ORGANIZATION_BLOCK OB 1
TITLE = "Main Program Sweep (Cycle)"
AUTHOR : Kng
NAME : Main
VERSION : 0.1
VAR_TEMP
  OB1_EV_CLASS : BYTE ;	//Bits 0-3 = 1 (Coming event), Bits 4-7 = 1 (Event class 1)
  OB1_SCAN_1 : BYTE ;	//1 (Cold restart scan 1 of OB 1), 3 (Scan 2-n of OB 1)
  OB1_PRIORITY : BYTE ;	//Priority of OB Execution
  OB1_OB_NUMBR : BYTE ;	//1 (Organization block 1, OB1)
  OB1_RESERVED_1 : BYTE ;	//Reserved for system
  OB1_RESERVED_2 : BYTE ;	//Reserved for system
  OB1_PREV_CYCLE : INT ;	//Cycle time of previous OB1 scan (milliseconds)
  OB1_MIN_CYCLE : INT ;	//Minimum cycle time of OB1 (milliseconds)
  OB1_MAX_CYCLE : INT ;	//Maximum cycle time of OB1 (milliseconds)
  OB1_DATE_TIME : DATE_AND_TIME ;	//Date and time OB1 started
END_VAR
BEGIN
NETWORK
TITLE =
//Strefy :
//skaner przod
//S-Srodek
//G-gora(spedycja)
//
//360-strefa 2 (GS)
//2123-strefa 1(GSD)
//11208-2(GS)
//17550-3(SD)
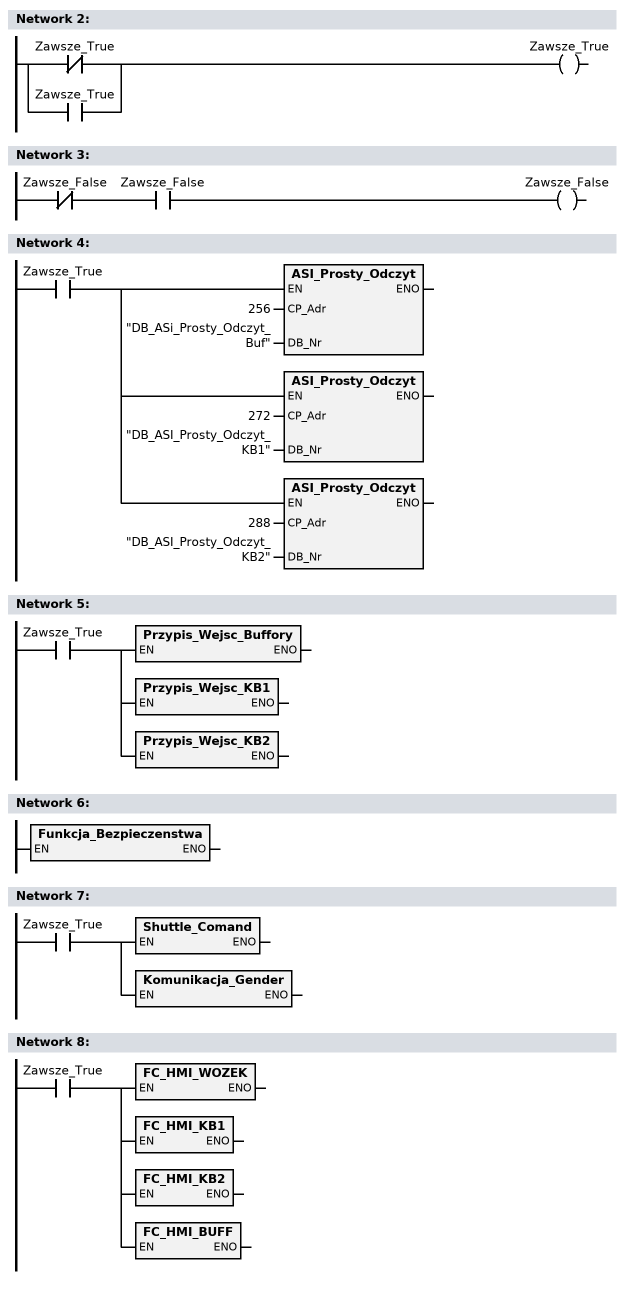
NETWORK
TITLE =
//Marki globalne
      ON    "Zawsze_True";
      O     "Zawsze_True";
      =     "Zawsze_True";
NETWORK
TITLE =
//Zawsze false
      AN    "Zawsze_False";
      A     "Zawsze_False";
      =     "Zawsze_False";
NETWORK
TITLE =
//Odczyt wejsc Asi
      A     "Zawsze_True";
      =     L 20.0;
      A     L 20.0;
      JNB   _001;
      CALL  "ASI_Prosty_Odczyt" (
           CP_Adr                   := 256,
           DB_Nr                    := "DB_ASi_Prosty_Odczyt_Buf");
_001: NOP   0;
      A     L 20.0;
      JNB   _002;
      CALL  "ASI_Prosty_Odczyt" (
           CP_Adr                   := 272,
           DB_Nr                    := "DB_ASI_Prosty_Odczyt_KB1");
_002: NOP   0;
      A     L 20.0;
      JNB   _003;
      CALL  "ASI_Prosty_Odczyt" (
           CP_Adr                   := 288,
           DB_Nr                    := "DB_ASI_Prosty_Odczyt_KB2");
_003: NOP   0;
NETWORK
TITLE =
//Przypisanie wejsc
      A     "Zawsze_True";
      =     L 20.0;
      A     L 20.0;
      JNB   _004;
      CALL  "Przypis_Wejsc_Buffory";
_004: NOP   0;
      A     L 20.0;
      JNB   _005;
      CALL  "Przypis_Wejsc_KB1";
_005: NOP   0;
      A     L 20.0;
      JNB   _006;
      CALL  "Przypis_Wejsc_KB2";
_006: NOP   0;
NETWORK
TITLE =
//Sterownie Reczny Auto
      CALL  "Funkcja_Bezpieczenstwa";
      NOP   0;
NETWORK
TITLE =
      A     "Zawsze_True";
      =     L 20.0;
      A     L 20.0;
      JNB   _007;
      CALL  "Shuttle_Comand";
_007: NOP   0;
      A     L 20.0;
      JNB   _008;
      CALL  "Komunikacja_Gender";
_008: NOP   0;
NETWORK
TITLE =
      A     "Zawsze_True";
      =     L 20.0;
      A     L 20.0;
      JNB   _009;
      CALL  "FC_HMI_WOZEK";
_009: NOP   0;
      A     L 20.0;
      JNB   _00a;
      CALL  "FC_HMI_KB1";
_00a: NOP   0;
      A     L 20.0;
      JNB   _00b;
      CALL  "FC_HMI_KB2";
_00b: NOP   0;
      A     L 20.0;
      JNB   _00c;
      CALL  "FC_HMI_BUFF";
_00c: NOP   0;
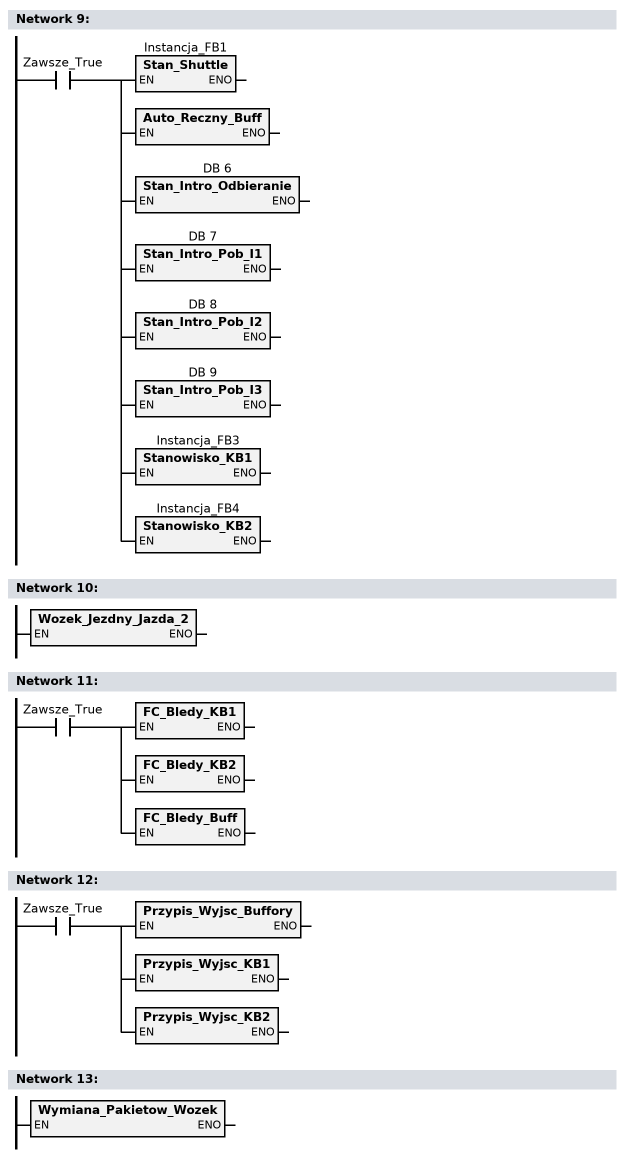
NETWORK
TITLE =
      A     "Zawsze_True";
      =     L 20.0;
      A     L 20.0;
      JNB   _00d;
      CALL  "Stan_Shuttle" , "Instancja_FB1";
_00d: NOP   0;
      A     L 20.0;
      JNB   _00e;
      CALL  "Auto_Reczny_Buff";
_00e: NOP   0;
      A     L 20.0;
      JNB   _00f;
      CALL  "Stan_Intro_Odbieranie" , DB 6;
_00f: NOP   0;
      A     L 20.0;
      JNB   _010;
      CALL  "Stan_Intro_Pob_I1" , DB 7;
_010: NOP   0;
      A     L 20.0;
      JNB   _011;
      CALL  "Stan_Intro_Pob_I2" , DB 8;
_011: NOP   0;
      A     L 20.0;
      JNB   _012;
      CALL  "Stan_Intro_Pob_I3" , DB 9;
_012: NOP   0;
      A     L 20.0;
      JNB   _013;
      CALL  "Stanowisko_KB1" , "Instancja_FB3";
_013: NOP   0;
      A     L 20.0;
      JNB   _014;
      CALL  "Stanowisko_KB2" , "Instancja_FB4";
_014: NOP   0;
NETWORK
TITLE =
      CALL  "Wozek_Jezdny_Jazda_2";
      NOP   0;
NETWORK
TITLE =
//Funcje bledow
      A     "Zawsze_True";
      =     L 20.0;
      A     L 20.0;
      JNB   _015;
      CALL  "FC_Bledy_KB1";
_015: NOP   0;
      A     L 20.0;
      JNB   _016;
      CALL  "FC_Bledy_KB2";
_016: NOP   0;
      A     L 20.0;
      JNB   _017;
      CALL  "FC_Bledy_Buff";
_017: NOP   0;
NETWORK
TITLE =
//Przypisanie wyjsc
//
      A     "Zawsze_True";
      =     L 20.0;
      A     L 20.0;
      JNB   _018;
      CALL  "Przypis_Wyjsc_Buffory";
_018: NOP   0;
      A     L 20.0;
      JNB   _019;
      CALL  "Przypis_Wyjsc_KB1";
_019: NOP   0;
      A     L 20.0;
      JNB   _01a;
      CALL  "Przypis_Wyjsc_KB2";
_01a: NOP   0;
NETWORK
TITLE =
      CALL  "Wymiana_Pakietow_Wozek";
      NOP   0;
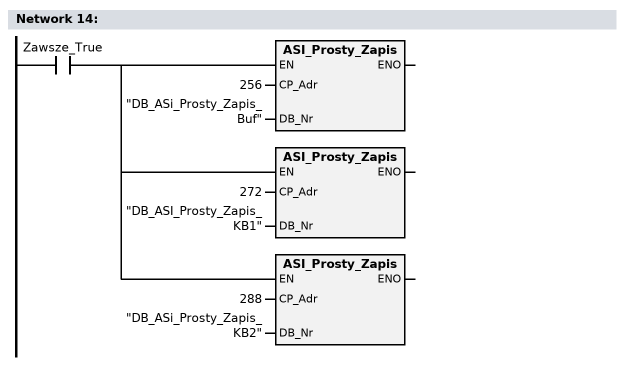
NETWORK
TITLE =
//Przypisanie Wyjsc Asi
      A     "Zawsze_True";
      =     L 20.0;
      A     L 20.0;
      JNB   _01b;
      CALL  "ASI_Prosty_Zapis" (
           CP_Adr                   := 256,
           DB_Nr                    := "DB_ASi_Prosty_Zapis_Buf");
_01b: NOP   0;
      A     L 20.0;
      JNB   _01c;
      CALL  "ASI_Prosty_Zapis" (
           CP_Adr                   := 272,
           DB_Nr                    := "DB_ASI_Prosty_Zapis_KB1");
_01c: NOP   0;
      A     L 20.0;
      JNB   _01d;
      CALL  "ASI_Prosty_Zapis" (
           CP_Adr                   := 288,
           DB_Nr                    := "DB_ASi_Prosty_Zapis_KB2");
_01d: NOP   0;
NETWORK
TITLE =
END_ORGANIZATION_BLOCK

ORGANIZATION_BLOCK "I/O_FLT1"	// OB 82
TITLE = "I/O Point Fault"
VERSION : 0.1
VAR_TEMP
  OB82_EV_CLASS : BYTE ;	//16#39, Event class 3, Entering event state, Internal fault event
  OB82_FLT_ID : BYTE ;	//16#XX, Fault identifcation code
  OB82_PRIORITY : BYTE ;	//Priority of OB Execution
  OB82_OB_NUMBR : BYTE ;	//82 (Organization block 82, OB82)
  OB82_RESERVED_1 : BYTE ;	//Reserved for system
  OB82_IO_FLAG : BYTE ;	//Input (01010100), Output (01010101)
  OB82_MDL_ADDR : WORD ;	//Base address of module with fault
  OB82_MDL_DEFECT : BOOL ;	//Module defective
  OB82_INT_FAULT : BOOL ;	//Internal fault
  OB82_EXT_FAULT : BOOL ;	//External fault
  OB82_PNT_INFO : BOOL ;	//Point information
  OB82_EXT_VOLTAGE : BOOL ;	//External voltage low
  OB82_FLD_CONNCTR : BOOL ;	//Field wiring connector missing
  OB82_NO_CONFIG : BOOL ;	//Module has no configuration data
  OB82_CONFIG_ERR : BOOL ;	//Module has configuration error
  OB82_MDL_TYPE : BYTE ;	//Type of module
  OB82_SUB_MDL_ERR : BOOL ;	//Sub-Module is missing or has error
  OB82_COMM_FAULT : BOOL ;	//Communication fault
  OB82_MDL_STOP : BOOL ;	//Module is stopped
  OB82_WTCH_DOG_FLT : BOOL ;	//Watch dog timer stopped module
  OB82_INT_PS_FLT : BOOL ;	//Internal power supply fault
  OB82_PRIM_BATT_FLT : BOOL ;	//Primary battery is in fault
  OB82_BCKUP_BATT_FLT : BOOL ;	//Backup battery is in fault
  OB82_RESERVED_2 : BOOL ;	//Reserved for system
  OB82_RACK_FLT : BOOL ;	//Rack fault, only for bus interface module
  OB82_PROC_FLT : BOOL ;	//Processor fault
  OB82_EPROM_FLT : BOOL ;	//EPROM fault
  OB82_RAM_FLT : BOOL ;	//RAM fault
  OB82_ADU_FLT : BOOL ;	//ADU fault
  OB82_FUSE_FLT : BOOL ;	//Fuse fault
  OB82_HW_INTR_FLT : BOOL ;	//Hardware interupt input in fault
  OB82_RESERVED_3 : BOOL ;	//Reserved for system
  OB82_DATE_TIME : DATE_AND_TIME ;	//Date and time OB82 started
END_VAR
BEGIN
NETWORK
TITLE =
END_ORGANIZATION_BLOCK

ORGANIZATION_BLOCK "RACK_FLT"	// OB 86
TITLE = "Loss Of Rack Fault"
VERSION : 0.1
VAR_TEMP
  OB86_EV_CLASS : BYTE ;	//16#38/39 Event class 3
  OB86_FLT_ID : BYTE ;	//16#C1/C4/C5, Fault identifcation code
  OB86_PRIORITY : BYTE ;	//Priority of OB Execution
  OB86_OB_NUMBR : BYTE ;	//86 (Organization block 86, OB86)
  OB86_RESERVED_1 : BYTE ;	//Reserved for system
  OB86_RESERVED_2 : BYTE ;	//Reserved for system
  OB86_MDL_ADDR : WORD ;	//Base address of IM module in rack with fault
  OB86_RACKS_FLTD : ARRAY  [0 .. 31 ] OF BOOL ;	//Racks in fault
  OB86_DATE_TIME : DATE_AND_TIME ;	//Date and time OB86 started
END_VAR
BEGIN
// (block stored without names or comments; labels and parameter names are numbered)
END_ORGANIZATION_BLOCK

ORGANIZATION_BLOCK "COMM_FLT"	// OB 87
TITLE = "Communication Fault"
VERSION : 0.1
VAR_TEMP
  OB87_EV_CLASS : BYTE ;	//16#39 Event class 3
  OB87_FLT_ID : BYTE ;	//16#XX, Fault identifcation code
  OB87_PRIORITY : BYTE ;	//Priority of OB Execution
  OB87_OB_NUMBR : BYTE ;	//87 (Organization block 87, OB87)
  OB87_RESERVED_1 : BYTE ;	//Reserved for system
  OB87_RESERVED_2 : BYTE ;	//Reserved for system
  OB87_RESERVED_3 : WORD ;	//Reserved for system
  OB87_RESERVED_4 : DWORD ;	//Reserved for system
  OB87_DATE_TIME : DATE_AND_TIME ;	//Date and time OB87 started
END_VAR
BEGIN
// (block stored without names or comments; labels and parameter names are numbered)
END_ORGANIZATION_BLOCK

ORGANIZATION_BLOCK "PROG_ERR"	// OB 121
TITLE = "Programming Error"
VERSION : 0.1
VAR_TEMP
  OB121_EV_CLASS : BYTE ;	//16#25, Event class 2, Entering event state, Internal fault event
  OB121_SW_FLT : BYTE ;	//16#XX Software programming fault
  OB121_PRIORITY : BYTE ;	//Priority of OB Execution
  OB121_OB_NUMBR : BYTE ;	//121 (Organization block 121, OB121)
  OB121_BLK_TYPE : BYTE ;	//16#88/8A/8B/8C/8E Type of block fault occured in
  OB121_RESERVED_1 : BYTE ;	//Reserved for system
  OB121_FLT_REG : WORD ;	//16#XX Specific register that caused fault
  OB121_BLK_NUM : WORD ;	//Number of block that programming fault occured in
  OB121_PRG_ADDR : WORD ;	//Address in block where programming fault occured
  OB121_DATE_TIME : DATE_AND_TIME ;	//Date and time OB121 started
END_VAR
BEGIN
NETWORK
TITLE =
END_ORGANIZATION_BLOCK

ORGANIZATION_BLOCK "MOD_ERR"	// OB 122
TITLE = "Module Access Error"
VERSION : 0.1
VAR_TEMP
  OB122_EV_CLASS : BYTE ;	//16#29, Event class 2, Entering event state, Internal fault event
  OB122_SW_FLT : BYTE ;	//16#XX Software error code
  OB122_PRIORITY : BYTE ;	//Priority of OB Execution
  OB122_OB_NUMBR : BYTE ;	//122 (Organization block 122, OB122)
  OB122_BLK_TYPE : BYTE ;	//16#88/8C/8E Type of block fault occured in
  OB122_MEM_AREA : BYTE ;	//Memory area where access error occured
  OB122_MEM_ADDR : WORD ;	//Memory address where access error occured
  OB122_BLK_NUM : WORD ;	//Block number in which error occured
  OB122_PRG_ADDR : WORD ;	//Program address where error occured
  OB122_DATE_TIME : DATE_AND_TIME ;	//Date and time OB1 started
END_VAR
BEGIN
// (block stored without names or comments; labels and parameter names are numbered)
END_ORGANIZATION_BLOCK

SYMBOL_TABLE
""		
"Instancja_FB1"	DB 1	FB 1
"Instancja_FB3"	DB 3	FB 3
"Instancja_FB4"	DB 4	FB 4
"DB_CONECTOR"	DB 10	DB 10	// Blok porzadkujacy czujniki lini
"DB_CONECTOR_KB1"	DB 11	DB 11
"DB_CONECTOR_KB2"	DB 12	DB 12
"DB_CONNECTOR_BUFF"	DB 13	DB 13
"DB_CONNECTOR_GEN"	DB 14	DB 14
"Asi_input"	DB 80	DB 80
"Asi_output"	DB 81	DB 81
"DB_ASI_Prosty_Odczyt_KB1"	DB 82	DB 82	// KB1
"DB_ASI_Prosty_Zapis_KB1"	DB 83	DB 83
"DB_ASI_Prosty_Odczyt_KB2"	DB 84	DB 84
"DB_ASi_Prosty_Zapis_KB2"	DB 85	DB 85
"DB_ASi_Prosty_Odczyt_Buf"	DB 86	DB 86	// Odczyt buffory
"DB_ASi_Prosty_Zapis_Buf"	DB 87	DB 87	// Asi db buffory
"Bledy_Shuttle"	DB 116	DB 116
"Bledy_KB1"	DB 117	DB 117
"Bledy_KB2"	DB 118	DB 118
"Bledy_Buffor"	DB 119	DB 119
"DB_HMI_KB1"	DB 121	DB 121
"DB_HMI_KB2"	DB 122	DB 122
"DB_HMI_BUF"	DB 123	DB 123
"DB_HMI_Wozek"	DB 128	DB 128
"COM_SHUTTLE"	DB 200	DB 200	// Blok komunikacji odbieranie shuttle
"LLOUT"	DB 201	DB 201
"LLIN"	DB 202	DB 202	// Blok wymiany danych dlugi
"COM_GENDER"	DB 205	DB 205
"Stale_Maszynowe"	DB 300	DB 300
"DB_Trace"	DB 402	DB 402
"Key_DB"	DB 409	DB 409
"Blok_Default"	DB 800	DB 800
"Blok_Write"	DB 801	DB 801
"Blok_Read"	DB 802	DB 802
"Def_Blok_Para_Wozek"	DB 811	DB 811
"Def_Blok_Kier_KB1"	DB 820	DB 820	// Blok stref kierunek KB1
"Def_Blok_Kier_Rot"	DB 821	DB 821
"Buffor_Rejestr"	DB 823	DB 823
"Buffor_Rejestr_HMI"	DB 824	DB 824
"Def_Stale_Maszynowe"	DB 830	DB 830
"Buffor_Kolejka"	DB 1123	DB 1123
"Blok_Def_Parametry"	DB 1701	DB 1701	// Blok Defaultowy parametrow
"Blok_Parametrow"	DB 1702	DB 1702
"Blok_Def_Kier_KB1"	DB 1720	DB 1720
"Blok_Def_Kier_Rot"	DB 1721	DB 1721
"Stan_Shuttle"	FB 1	FB 1
"Stanowisko_KB1"	FB 3	FB 3	// Stanowisko Kolbus 1
"Stanowisko_KB2"	FB 4	FB 4	// Stanowisko Kolbus 2
"Blok_Jazdy_Band"	FB 5	FB 5
"Stan_Intro_Odbieranie"	FB 6	FB 6
"Stan_Intro_Pob_I1"	FB 7	FB 7
"Stan_Intro_Pob_I2"	FB 8	FB 8	// Stanowisko wozek jezdny
"Stan_Intro_Pob_I3"	FB 9	FB 9
"FB_Uzbrajanie"	FB 10	FB 10	// Funkcja uzbrajanie\
"Filtr_zbocza_2"	FB 14	FB 14
"T_ON"	FB 20	FB 20	// Timer on delay with memory
"T_ON_+_RESET"	FB 21	FB 21	// Czasowka on delay z zapamietanym czasem  + reset
"Banda_Pojedyncza"	FB 30	FB 30
"Banda_Obr_1"	FB 31	FB 31	// Banda obrotowa o dwoch wlotach i jednej fotokomorce
"Band_Wozka"	FB 32	FB 32	// Banda wozka z trybem recznym
"Banda_Poj_+_Tryb_Reczny"	FB 33	FB 33
"B_Obr_+_Reczny"	FB 35	FB 35
"Banda_Obr_+_Reczny"	FB 36	FB 36	// Banda obrotwa + reczny
"Banda_Poj_+_Winda"	FB 37	FB 37	// Banda pojedyncza + winda + tryb reczny
"Wybranie_Wjazdu"	FB 50	FB 50
"Obr_Na_Poz_1"	FB 51	FB 51
"Pozycjonowanie_Bandy"	FB 55	FB 55
"Obr_Na_Poz_1_Pelny"	FB 61	FB 61
"KB2_Reczny"	FC 1	FC 1
"Funkcja_Bezpieczenstwa"	FC 3	FC 3
"Oryginalna_FC3"	FC 4	FC 4
"Wozek_Jezdny_Jazda"	FC 5	FC 5
"Wozek_Jezdny_Jazda_2"	FC 6	FC 6	// Funkcja sterujaca lampkami
"Sprawdzenie_Okna"	FC 7	FC 7	// Sprawdzenie czy wartosc miesci sie w oknie
"Lenze_Sew_Shell_KB1"	FC 8	FC 8
"Lenze_Sew_Shell_KB2"	FC 9	FC 9	// Nakladka na falownik Lenze by czytac jak Sewa
"Fal_Lenze_V_3"	FC 10	FC 10
"Przyciski_Dwufunkcyjne"	FC 11	FC 11
"Sterowanie_Ramp"	FC 12	FC 12
"Auto_Reczny_KB1"	FC 13	FC 13
"Auto_Reczny_KB2"	FC 14	FC 14
"Auto_Reczny_Buff"	FC 15	FC 15
"Przyporzadkowanie_Wejsc"	FC 20	FC 20
"Przyporzadkowanie_Wyjsc"	FC 21	FC 21
"Przypis_Wejsc_KB1"	FC 22	FC 22
"Przypis_Wyjsc_KB1"	FC 23	FC 23
"Przypis_Wejsc_KB2"	FC 24	FC 24
"Przypis_Wyjsc_KB2"	FC 25	FC 25
"Przypis_Wejsc_Buffory"	FC 26	FC 26
"Przypis_Wyjsc_Buffory"	FC 27	FC 27
"Rejestr_Tasm"	FC 30	FC 30
"qqq"	FC 31	FC 31
"Ruch_Palety"	FC 40	FC 40
"Ruch_Palety_Winda"	FC 41	FC 41	// Kasowanie_Bledow
"Wybor_Wjazdu"	FC 50	FC 50	// Wybor miejsca pobierania palety
"Obrotnica_Na_Pozycje"	FC 51	FC 51
"LT_BT"	FC 62	FC 62	// Convert local time to base time
"ASI_Odczyt"	FC 80	FC 80
"ASI_Zapis"	FC 81	FC 81
"ASI_Prosty_Odczyt"	FC 82	FC 82	// Prosty odczyt modulow asi- nasjszybsza wersja
"ASI_Prosty_Zapis"	FC 83	FC 83	// Prosty zapis danych do modulow Asi (nastawiony na predkosc)
"Opoznienie_Wylotu"	FC 85	FC 85
"FC_Bledy_KB1"	FC 117	FC 117
"FC_Bledy_KB2"	FC 118	FC 118
"FC_Bledy_Buff"	FC 119	FC 119
"FC_HMI_KB1"	FC 121	FC 121
"FC_HMI_KB2"	FC 122	FC 122
"FC_HMI_BUFF"	FC 123	FC 123
"FC_HMI_WOZEK"	FC 128	FC 128
"Funkcja_Zegara"	FC 140	FC 140	// Funkcja zegara
"Shuttle_Comand"	FC 200	FC 200
"Wymiana_Pakietow_Wozek"	FC 201	FC 201	// Wymiana duzej ilosci danych z wozkiem
"Komunikacja_Gender"	FC 205	FC 205
"Monitor_Bandy"	FC 313	FC 313	// Funkcja monitorujaca przejezdzajacy produkt
"Monitor_Bandy_2"	FC 314	FC 314	// Monitor Bandy z wykryciem auto
"Monitor_Bandy_+_Reczny"	FC 315	FC 315	// Funkcja monitorujaca + tryb reczny
"Monitor_Palety"	FC 316	FC 316	// Auto wyszukiwanie palety w masce
"Znajdz_Widmo"	FC 317	FC 317	// Funkcja szuka palety widmo
"Dekoduj_Maske"	FC 320	FC 320
"Dobor_Elementow_Lini"	FC 400	FC 400
"Opis_Dwubajtu_Zadanego"	FC 401	FC 401
"Sorting_FC"	FC 402	FC 402
"Shuttle_Queue"	FC 403	FC 403
"Wozek_Queue_V2"	FC 404	FC 404
"Sorting_V2"	FC 405	FC 405
"Wozek_Queue_V3"	FC 408	FC 408
"Sorting_V3"	FC 409	FC 409
"FC_Nawigator"	FC 410	FC 410
"Wozek_Jezdny_Kolejka"	FC 600	FC 600
"Send_Data"	FC 700	FC 700
"Receive_Data"	FC 701	FC 701
"Read_Data"	FC 702	FC 702
"Share_Data"	FC 703	FC 703	// Funkcja udostepniajaca dane
"Ekran_Para_Wozek"	FC 1701	FC 1701
"Ekran_Kier_KB1"	FC 1720	FC 1720
"Ekran_Kier_Rot"	FC 1721	FC 1721
"Ekran_Para_Odbieranie"	FC 1730	FC 1730
"PB_Strefa"	I 4.0	BOOL
"PB_Funkcja"	I 4.3	BOOL
"Obrtonica_Tyl"	I 5.1	BOOL
"Buff_PB_Reset_Przek_Bezp"	I 8.0	BOOL
"Buff_PB_Semi_Auto"	I 8.1	BOOL
"Buff_PB_Auto"	I 8.2	BOOL
"i_Buff_PB_Zal_Wozka"	I 8.3	BOOL
"Buff_Foto_Wozek_Pob"	I 8.7	BOOL
"Buff_Przek_Bezp_Ok"	I 10.0	BOOL
"Buff_Przek_Shuttle_OK"	I 10.1	BOOL
"KB1_PB_Reset_Bezp"	I 12.0	BOOL	// Przycisk kasowanie strefy bezpieczenstwa
"KB1_PB_Semi_Auto"	I 12.1	BOOL	// Przycisk polautomatyki
"KB1_PB_Auto"	I 12.2	BOOL	// Przycisk Automatyki
"KB1_PB_Funkcja"	I 12.3	BOOL
"KB1_PB_Shuttle_Tyl"	I 12.4	BOOL	// Przycisk shuttle przod
"KB1_PB_Shuttle_Przod"	I 12.5	BOOL	// Przycisk shuttle tyl
"KB1_PB_Winda_Przod"	I 12.6	BOOL	// Przycisk winda przod
"KB1_PB_Winda_Tyl"	I 12.7	BOOL	// Przycisk winda tyl
"KB1_PB_Obrotnica_Przod"	I 13.0	BOOL
"KB1_PB_Obrotnica_Tyl"	I 13.1	BOOL
"KB1_PB_Band_Seg_Przod"	I 13.2	BOOL	// Banda Segbetr przod
"KB1_PB_Band_Seg_Tyl"	I 13.3	BOOL	// Banda Segbert tyl
"KB1_PB_WWylot_2_Przod"	I 13.4	BOOL
"KB1_PB_WWylot_2_Tyl"	I 13.5	BOOL
"KB1_Rez_I23.6"	I 13.6	BOOL
"KB1_Rez_I23.7"	I 13.7	BOOL
"KB1_P_Bezp_Ok"	I 14.0	BOOL	// Przekaznik bezpieczenstwa ok
"KB1_P_Bezp_Shuttle_Ok"	I 14.1	BOOL	// Przekanik bezpieczenstwa Shuttle ok
"KB1_Petla_Fuse_Ok"	I 14.2	BOOL	// Petla bezpiecznikow Ok
"KB1_PB_Wyb_Obr_Lewo"	I 14.3	BOOL
"KB1_PB_Wyb_Obr_Prawo"	I 14.4	BOOL
"KB1_PB_Grzybek_Pracy"	I 14.5	BOOL
"KB1_PB_Pedal_Pracy_1"	I 14.6	BOOL
"KB1_PB_Pedal_Pracy_2"	I 14.7	BOOL
"KB1_Winda_W_Dole"	I 15.0	BOOL
"KB1_Winda_W_Gorze"	I 15.1	BOOL
"KB1_Foto_Shuttle"	I 15.2	BOOL
"KB1_Obecn_Wozka_Wylot_2"	I 15.3	BOOL
"KB1_Rezerwa_I25.4"	I 15.4	BOOL
"KB1_Rezerwa_I25.5"	I 15.5	BOOL
"KB1_Rezerwa_I25.6"	I 15.6	BOOL
"KB1_Rezerwa_I25.7"	I 15.7	BOOL
"KB1_Foto_Seg_Przod"	I 16.0	BOOL
"KB1_Foto_Segbert_Tyl"	I 16.1	BOOL
"KB1_Zasilanie_Seg_Fal"	I 16.2	BOOL	// Falowniki sa zasilane
"KB1_Obr_Foto_2"	I 17.0	BOOL
"KB1_Obr_Foto_1"	I 17.1	BOOL
"KB2_PB_Reset_Bezp"	I 22.0	BOOL	// Przycisk kasowanie strefy bezpieczenstwa
"KB2_PB_Semi_Auto"	I 22.1	BOOL	// Przycisk polautomatyki
"KB2_PB_Auto"	I 22.2	BOOL	// Przycisk Automatyki
"KB2_PB_Funkcja"	I 22.3	BOOL
"KB2_PB_Shuttle_Tyl"	I 22.4	BOOL	// Przycisk shuttle przod
"KB2_PB_Shuttle_Przod"	I 22.5	BOOL	// Przycisk shuttle tyl
"KB2_PB_Winda_Przod"	I 22.6	BOOL	// Przycisk winda przod
"KB2_PB_Winda_Tyl"	I 22.7	BOOL	// Przycisk winda tyl
"KB2_PB_Obrotnica_Przod"	I 23.0	BOOL
"KB2_PB_Obrotnica_Tyl"	I 23.1	BOOL
"KB2_PB_Band_Seg_Przod"	I 23.2	BOOL	// Banda Segbetr przod
"KB2_PB_Band_Seg_Tyl"	I 23.3	BOOL	// Banda Segbert tyl
"KB2_PB_WWylot_2_Przod"	I 23.4	BOOL
"KB2_PB_WWylot_2_Tyl"	I 23.5	BOOL
"KB2_Rez_I23.6"	I 23.6	BOOL
"KB2_Rez_I23.7"	I 23.7	BOOL
"KB2_P_Bezp_Ok"	I 24.0	BOOL	// Przekaznik bezpieczenstwa ok
"KB2_P_Bezp_Shuttle_Ok"	I 24.1	BOOL	// Przekanik bezpieczenstwa Shuttle ok
"KB2_Petla_Fuse_Ok"	I 24.2	BOOL	// Petla bezpiecznikow Ok
"KB2_PB_Wyb_Obr_Lewo"	I 24.3	BOOL
"KB2_PB_Wyb_Obr_Prawo"	I 24.4	BOOL
"KB2_PB_Grzybek_Pracy"	I 24.5	BOOL
"KB2_PB_Pedal_Pracy_1"	I 24.6	BOOL
"KB2_PB_Pedal_Pracy_2"	I 24.7	BOOL
"KB2_Winda_W_Dole"	I 25.0	BOOL
"KB2_Winda_W_Gorze"	I 25.1	BOOL
"KB2_Foto_Shuttle"	I 25.2	BOOL
"KB2_Obecn_Wozka_Wylot_2"	I 25.3	BOOL
"KB2_Rezerwa_I25.4"	I 25.4	BOOL
"KB2_Rezerwa_I25.5"	I 25.5	BOOL
"KB2_Rezerwa_I25.6"	I 25.6	BOOL
"KB2_Rezerwa_I25.7"	I 25.7	BOOL
"KB2_Foto_Seg_Przod"	I 26.0	BOOL
"KB2_Foto_Banda_Seg_Tyl"	I 26.1	BOOL
"KB2_Zasilanie_Seg_Fal"	I 26.2	BOOL
"KB2_Obr_Foto_2"	I 27.0	BOOL
"KB2_Obr_Foto_1"	I 27.1	BOOL
"ip_Bit_Kom_Shuttle"	I 30.0	BOOL	// bit komunikacji ( Shuttle <---)
"ip_Potw_Nowej_Pozycji"	I 31.1	BOOL	// Bit potwierdzenia przyjecia nowej pozycji (Shuttle <---)
"ip_Shuttle_Na_Pozycji"	I 31.2	BOOL	// Wozek na pozycji (Shuttle <--)
"ip_Shuttle_Stoi"	I 31.3	BOOL	// Wozek nie jedzie (Shuttle <--)
"ip_Potw_Zasprz"	I 31.4	BOOL	// Potwierdzenie zasprzeglenia (Shuttle <--)
"ip_Potw_Rozprz"	I 31.5	BOOL	// Potwierdzenie Rozprzeglenia (Shuttle <--)
"ip_Foto_Przod"	I 31.6	BOOL	// Fotokomorka wozek przod (Shuttle <--)
"ip_Foto_Wozek_Tyl"	I 31.7	BOOL	// Fotokomorka wozek tyl (Shuttle <--)
"Buff_2_PB_Reset_Przek_B"	I 80.0	BOOL
"Buff_2_PB_Semi_Auto"	I 80.1	BOOL
"Buff_2_PB_Auto"	I 80.2	BOOL
"Buff_2_PB_Banda_7_Lewo"	I 81.0	BOOL
"Buff_2_PB_Banda_7_Prawo"	I 81.1	BOOL
"Buff_2_PB_Banda_8_Lewo"	I 81.2	BOOL
"Buff_2_PB_Banda_8_Prawo"	I 81.3	BOOL
"Buff_2_PB_Banda_17_Lewo"	I 81.4	BOOL
"Buff_2_PB_Banda_17_Prawo"	I 81.5	BOOL
"Buff_2_PB_Banda_18_Lewo"	I 81.6	BOOL
"Buff_2_PB_Banda_18_Prawo"	I 81.7	BOOL
"Buff_2_PB_Banda_W_Lewo"	I 82.0	BOOL
"Buff_2_PB_Banda_W_Prawo"	I 82.1	BOOL
"Buff_2_Foto_Wlot_2"	I 82.2	BOOL
"Buff_2_Foto_Wlot_3"	I 82.3	BOOL
"Dword_0_Shuttle"	ID 30	DWORD
"ip_Poz_Akt_Wozka"	ID 34	DINT	// Pozycja aktualna wozka (Shuttle <--)
"Zawsze_True"	M 0.0	BOOL
"Zawsze_False"	M 0.1	BOOL
"Marka_X"	M 0.3	BOOL	// Marka output wszystko jedno
"Help_Start"	M 1.0	BOOL
"Help_Zbocze_Start"	M 1.1	BOOL
"Help_Start_2"	M 1.2	BOOL
"Marka_Bezpieczenstwa_0"	M 2.0	BOOL	// Marka_Bezpieczenstwa poziomu 0
"Marka_Start_Stop"	M 2.1	BOOL
"Marka_Bezpieczenstwa_2"	M 2.2	BOOL
"Rejon_Bindownicy_Stop"	M 2.3	BOOL
"Strefa_Bind_Ok"	M 2.4	BOOL
"Help_PB_Stop"	M 2.5	BOOL
"Edge_2_6"	M 2.6	BOOL
"Freeze"	M 2.7	BOOL
"Brak_Bledu"	M 3.0	BOOL
"Falowniki_OK"	M 3.1	BOOL
"Fuse_OK"	M 3.2	BOOL
"Help_Freeze"	M 3.3	BOOL
"Marka_Bezpieczenstwa_3"	M 3.4	BOOL
"Zezwolenie_Na_Wjazd"	M 3.5	BOOL	// Do stawiania lini
"Stop_Hmi"	M 3.7	BOOL
"Jedz_Na_Nowa_Pozycje"	M 20.0	BOOL
"Edge_M20.1"	M 20.1	BOOL
"Brak_Komunikacji_Shuttle"	M 20.2	BOOL
"Shuttle_Na_Pozycji"	M 20.3	BOOL	// Shuttle jest na pozycji zadanej
"Pozycja_Gorna_Ok"	M 20.4	BOOL
"Pozycja_Dolna_Ok"	M 20.5	BOOL
"Reset zadania"	M 20.6	BOOL
"Edge_M20.7"	M 20.7	BOOL
"Zasprzegnij_Wozek"	M 21.0	BOOL
"Rozprzeglenie_Wozka"	M 21.1	BOOL
"Wozek_zasprzeglony"	M 21.2	BOOL
"Pom_Bit_Zasprzeg"	M 21.4	BOOL
"Foto_Wozek_Przod"	M 22.0	BOOL	// Fotokomorka wozek przod
"Foto_Wozek_Tyl"	M 22.1	BOOL	// Fotokomorka wozek tyl
"Silnik_Banda_Wozek_lewo"	M 22.2	BOOL
"Silnik_Banda_Wozke_Prawo"	M 22.3	BOOL
"Foto_Wozek_Przod_Opoz"	M 22.4	BOOL
"Foto_Wozek_Tyl_Opoz"	M 22.5	BOOL
"Bezpieczne_Pokrycie_Foto"	M 22.6	BOOL
"Zasprzeglenie_KB1"	M 23.0	BOOL	// Wozek zasprzeglony do KB1
"Zasprzeglenie_KB2"	M 23.1	BOOL	// Wozek zasprzeglony do KB2
"Zasprzeglenie_Pob_I1"	M 23.2	BOOL	// Zasprzeglenie Intro pobieranie
"Zasprzeglenie_Gender"	M 23.3	BOOL	// Wozek zasprzeglony do Gender
"Zasprzeglenie_Odbieranie"	M 23.4	BOOL	// Wozek zasprzeglony do odbierania
"Banda_Wozka_Pracuje"	M 23.5	BOOL
"Zasprzeglenie_Pob_I2"	M 23.6	BOOL
"Zasprzeglenie_Pob_I3"	M 23.7	BOOL
"Wozek_Marka_Bezp"	M 24.0	BOOL	// Marka Bezpieczenstwa wozek
"Wozek_Odwrocone_Sygnaly"	M 24.1	BOOL
"Wozek_Auto_Reczny"	M 24.2	BOOL	// Auto reczny wozek
"Wozek_Zez_Od_Nastepnej"	M 24.3	BOOL
"Wozek_Dost_Od_Nast"	M 24.4	BOOL	// Paleta dostarczona sygnal od nastepnej
"Wozek_Zabierz_Od_Pop"	M 24.5	BOOL	// Sygnal zabierz od poprzedniej
"Wozek_Zez_Reczny_Od_Pop"	M 24.6	BOOL	// Sygnal zezwolenia recznego od poprzedniej
"Wozek_Przycisk_Przod"	M 24.7	BOOL
"Wozek_Przycisk_Tyl"	M 25.0	BOOL
"Bit_Resetu_Interfejsu"	M 25.1	BOOL
"Wozek_Reczny_Od_Nast"	M 25.2	BOOL
"Wozek_Zabierz_Do_Nast"	M 26.0	BOOL	// Sygnal wozka zabierz do nastepnej
"Wozek_Zez_Do_Pop"	M 26.1	BOOL
"Wozek_Paleta_Dost_Do_Pop"	M 26.2	BOOL	// Paleta dostarczona do poprzedniej
"Wozek_Zez_Reczny_Do_Nast"	M 26.3	BOOL
"Wozek_Zez_Reczny_Do_Pop"	M 26.4	BOOL
"Wozek_Nieb_Zajetosc"	M 26.5	BOOL
"Help_Widmo"	M 27.0	BOOL
"Foto_Woz_Odbieranie"	M 27.1	BOOL	// Foto woz na odbieraniu
"Na_Pozycji_KB1"	M 40.0	BOOL
"Na_Pozycji_KB2"	M 40.1	BOOL
"Na_Pozycji_Gender"	M 40.2	BOOL
"Na_Pozycji_Odbieranie"	M 40.3	BOOL
"Na_Pozycji_Pob_I1"	M 40.4	BOOL
"Na_Pozycji_Pob_I2"	M 40.5	BOOL
"Na_Pozycji_Pob_I3"	M 40.6	BOOL
"Jedz_Na_KB1"	M 50.0	BOOL
"Jedz_Na_KB2"	M 50.1	BOOL
"Jedz_Na_Gender"	M 50.2	BOOL
"Jedz_Na_Odbior"	M 50.3	BOOL
"Jedz_Na_Pob_I1"	M 50.4	BOOL
"Jedz_Na_Zadana"	M 50.5	BOOL
"Marka_Jazdy_Na_Nowa_Poz"	M 50.6	BOOL
"Edge_50.7"	M 50.7	BOOL
"Edge_M51.0"	M 51.0	BOOL
"Blokada_Pobierania"	M 51.1	BOOL
"Jedz_Na_Pob_I2"	M 52.0	BOOL
"Jedz_Na_Pob_I3"	M 52.1	BOOL
"KB1_M_Bezpieczenstwa_0"	M 102.0	BOOL
"KB1_Auto_Reczny"	M 104.0	BOOL
"M106.0"	M 106.0	BOOL
"M106.1"	M 106.1	BOOL
"Zbocz_M106.2"	M 106.2	BOOL
"Zbocze_M106.3"	M 106.3	BOOL
"Warunek_Pustych_Kolbusow"	M 106.4	BOOL
"Zbocze_M106.5"	M 106.5	BOOL
"Paleta_Na_Pob_I1"	M 106.6	BOOL
"Blokuj_Pobieranie"	M 106.7	BOOL
"Edge_M107.0"	M 107.0	BOOL
"Edge_M107.1"	M 107.1	BOOL
"KB1_Tryb_Uzbr_Aktyw"	M 108.0	BOOL
"KB1_Bit_Ham_Sew"	M 110.0	BOOL
"KB1_Zez_Hand_Do_Nast"	M 110.1	BOOL
"KB1_M_Foto_Segbert"	M 111.0	BOOL
"KB1_Zab_od_Segbert"	M 111.1	BOOL
"KB1_B_Seg_Hand_Przod"	M 111.3	BOOL
"KB1_B_Seg_Auto_Przod"	M 111.4	BOOL
"KB1_Zezwolenie_Dla_Windy"	M 111.6	BOOL
"KB1_Warunki_Windy"	M 114.0	BOOL
"KB1_Warunki_Obrotnicy"	M 114.1	BOOL
"Edge_M114.2"	M 114.2	BOOL
"KB1_Wrunk_Przyjzd_Wozka"	M 114.3	BOOL
"KB1_Podwojny_Wlot"	M 120.0	BOOL	// 1-tak,0-nie
"KB1_Inline"	M 120.1	BOOL	// 1-tak,0-nie
"KB1_Uzbrajanie_Seg"	M 120.2	BOOL	// 1-tak,0-nie
"KB1_Uzbrajenie_Feedera"	M 120.3	BOOL	// 1-tak,0-nie
"KB1_Res_220_0_4"	M 120.4	BOOL
"KB1_Res_220_0_5"	M 120.5	BOOL
"KB1_Res_220_0_6"	M 120.6	BOOL
"KB1_Res_220_0_7"	M 120.7	BOOL
"KB1_VPB_Obrotnica_Przod"	M 121.0	BOOL	// VPB-virtual push button
"KB1_VPB_Obrotnica_Tyl"	M 121.1	BOOL	// VPB-virtual push button
"KB1_VPB_Obrotnica_CW"	M 121.2	BOOL	// VPB-virtual push button
"KB1_VPB_Obrotnica_CCW"	M 121.3	BOOL	// VPB-virtula push button
"KB1_Virutal_Foto_Wylot"	M 121.4	BOOL
"KB1_M121.5"	M 121.5	BOOL
"KB1_VPB_Winda_Przod"	M 122.0	BOOL
"KB1_VPB_Winda_Tyl"	M 122.1	BOOL
"KB1_VPB_Winda_Gora"	M 122.2	BOOL
"KB1_VPB_Winda_Dol"	M 122.3	BOOL
"KB1_Winda_Jazda_Gora"	M 122.4	BOOL
"KB1_Winda_Jazda_Dol"	M 122.5	BOOL
"KB1_Not_Aus_Pulpit_OK"	M 123.0	BOOL	// Not Aus adres 20 ok
"KB1_Grzyb_Bezp_OK"	M 123.1	BOOL	// Grzyb bezpieczenistwa Adres 21 OK
"KB1_Przek_Bezp_Potw"	M 123.3	BOOL	// Przekaznik bezpieczenstwa mozliwy do potwierdzenia
"KB1_Blada_Lini"	M 123.4	BOOL
"KB1_Uzbr_Oczek_Akt"	M 124.0	BOOL
"KB1_Start_Uzbr_Shot"	M 124.1	BOOL	// Krotki sygnal startu uzbrajania
"KB1_Sygnal_Kon_Uzbr"	M 124.2	BOOL	// Sygnal konca uzbrajania
"KB1_Pedal_W_Lewo"	M 124.3	BOOL	// Pedal obrotnicy jw lewo
"KB1_Pedal_W_Prawo"	M 124.4	BOOL	// Pedal obrotnicy jw prawo
"KB1_Uzbr_Aktywne"	M 124.5	BOOL	// Uzbrajanie palety jest aktywne
"KB1_Zez_Na_Uzbrajanie"	M 124.6	BOOL
"KB1_Uzbrj_Reczne"	M 124.7	BOOL
"KB1_Sygnal_Dzwiekowy"	M 125.0	BOOL
"KB1_Zbocze_M125.1"	M 125.1	BOOL
"KB1_Zez_Na_Uzbraj"	M 142.6	BOOL
"KB1_Help_Poz_1"	M 200.0	BOOL
"KB2_Help_Poz_1"	M 200.1	BOOL
"KB2_Help_Poz_2"	M 200.2	BOOL
"Buffory_Help_Poz_1"	M 200.3	BOOL
"Gender_Help_Poz_1"	M 200.4	BOOL
"Gender_Help_Poz_2"	M 200.5	BOOL
"KB2_M_Bezpieczenstwa_0"	M 202.0	BOOL
"KB2_Auto_Reczny"	M 204.0	BOOL	// 1-Auto,0-Reczny
"Edge_M207.0"	M 207.0	BOOL
"Edge_M207.1"	M 207.1	BOOL
"KB2_Tryb_Uzbr_Aktyw"	M 208.0	BOOL
"KB2_Bit_Ham_Sew"	M 210.0	BOOL
"KB2_Zez_Hand_Do_Nast"	M 210.1	BOOL
"KB2_M_Foto_Segbert"	M 211.0	BOOL
"KB2_Zab_od_Segbert"	M 211.1	BOOL
"KB2_B_Seg_Hand_Przod"	M 211.3	BOOL
"KB2_B_Seg_Auto_Przod"	M 211.4	BOOL
"KB2_Zezwolenie_Dla_Windy"	M 211.6	BOOL
"KB2_Warunki_Windy"	M 214.0	BOOL
"KB2_Warunki_Obrotnicy"	M 214.1	BOOL
"Edge_M214.2"	M 214.2	BOOL
"KB2_Wrunk_Przyjzd_Wozka"	M 214.3	BOOL
"KB2_Podwojny_Wlot"	M 220.0	BOOL	// 1-tak,0-nie
"KB2_Inline"	M 220.1	BOOL	// 1-tak,0-nie
"KB2_Uzbrajanie_Seg"	M 220.2	BOOL	// 1-tak,0-nie
"KB2_Uzbrajenie_Feedera"	M 220.3	BOOL	// 1-tak,0-nie
"KB2_Res_220_0_4"	M 220.4	BOOL
"KB2_Res_220_0_5"	M 220.5	BOOL
"KB2_Res_220_0_6"	M 220.6	BOOL
"KB2_Res_220_0_7"	M 220.7	BOOL
"KB2_VPB_Obrotnica_Przod"	M 221.0	BOOL	// VPB-virtual push button
"KB2_VPB_Obrotnica_Tyl"	M 221.1	BOOL	// VPB-virtual push button
"KB2_VPB_Obrotnica_CW"	M 221.2	BOOL	// VPB-virtual push button
"KB2_VPB_Obrotnica_CCW"	M 221.3	BOOL	// VPB-virtula push button
"KB2_Virutal_Foto_Wylot"	M 221.4	BOOL
"KB2_M221.5"	M 221.5	BOOL
"KB2_VPB_Winda_Przod"	M 222.0	BOOL
"KB2_VPB_Winda_Tyl"	M 222.1	BOOL
"KB2_VPB_Winda_Gora"	M 222.2	BOOL
"KB2_VPB_Winda_Dol"	M 222.3	BOOL
"KB2_Winda_Jazda_Gora"	M 222.4	BOOL
"KB2_Winda_Jazda_Dol"	M 222.5	BOOL
"KB2_Not_Aus_Pulpit_OK"	M 223.0	BOOL	// Not Aus adres 20 ok
"KB2_Grzyb_Bezp_OK"	M 223.1	BOOL	// Grzyb bezpieczenistwa Adres 21 OK
"KB2_Przek_Bezp_Potw"	M 223.3	BOOL	// Przekaznik bezpieczenstwa mozliwy do potwierdzenia
"KB2_Blada_Lini"	M 223.4	BOOL
"KB2_Uzbr_Oczek_Akt"	M 224.0	BOOL
"KB2_Start_Uzbr_Shot"	M 224.1	BOOL	// Krotki sygnal startu uzbrajania
"KB2_Sygnal_Kon_Uzbr"	M 224.2	BOOL	// Sygnal konca uzbrajania
"KB2_Pedal_W_Lewo"	M 224.3	BOOL	// Pedal obrotnicy jw lewo
"KB2_Pedal_W_Prawo"	M 224.4	BOOL	// Pedal obrotnicy jw prawo
"KB2_Uzbr_Aktywne"	M 224.5	BOOL	// Uzbrajanie palety jest aktywne
"KB2_Zez_Na_Uzbrajanie"	M 224.6	BOOL
"KB2_Uzbrj_Reczne"	M 224.7	BOOL
"KB2_Sygnal_Dzwiekowy"	M 225.0	BOOL
"KB2_Zbocze_M225.1"	M 225.1	BOOL
"Marka_Bezpieczenstwa_Buf"	M 302.0	BOOL
"Silniki_Sew_OK"	M 302.3	BOOL
"Help_M302.7"	M 302.7	BOOL
"I1_Buf_Auto_Reczny"	M 304.0	BOOL
"I1_Buff_Opoz_Startu"	M 304.2	BOOL
"I2_Buff_Opoz_Startu"	M 304.3	BOOL
"I3_Buff_Opoz_Startu"	M 304.4	BOOL
"I2_I3_Buf_Auto_Reczny"	M 305.0	BOOL
"Buff_Obwody_Got_Do_Potw"	M 306.0	BOOL
"Edge_M307.0"	M 307.0	BOOL
"Edge_M307.1"	M 307.1	BOOL
"M_Miganie_200ms"	M 310.0	BOOL
"M_Miganie_500ms"	M 310.1	BOOL
"M_Miganie_100ms"	M 310.2	BOOL
"I1_Kier_Pob_Spedycja"	M 311.0	BOOL
"I1_Kier_Pob_Intro"	M 311.1	BOOL
"I1_Buff_Wiaz_Pop"	M 311.2	BOOL
"I1_Buff_Wiaz_Wzdl"	M 311.3	BOOL
"Blokuj_Czerwone"	M 312.0	BOOL
"Buff_Opoz_Foto_Wylot"	M 313.0	BOOL
"Help_M313.1"	M 313.1	BOOL
"Buff_Odbier_Wolne"	M 314.0	BOOL	// Miejsce na buforach jest wolne
"I1_Buff_Kod_0"	M 315.0	BOOL
"I1_Buff_Kod_1"	M 315.1	BOOL
"I1_Buff_Kod_2"	M 315.2	BOOL
"I1_Buff_Kod_3"	M 315.3	BOOL
"Stanowisko_I1"	M 315.4	BOOL
"I1_Stan_Ma_Zadanie"	M 315.5	BOOL
"Edge_M315.6"	M 315.6	BOOL
"Help_M315.7"	M 315.7	BOOL
"I2_Kier_Pob_Spedycja"	M 317.0	BOOL
"I2_Kier_Pob_Intro"	M 317.1	BOOL
"I2_Buff_Wiaz_Pop"	M 317.2	BOOL
"I2_Buff_Wiaz_Wzdl"	M 317.3	BOOL
"I2_Buff_Kod_0"	M 318.0	BOOL
"I2_Buff_Kod_1"	M 318.1	BOOL
"I2_Buff_Kod_2"	M 318.2	BOOL
"I2_Buff_Kod_3"	M 318.3	BOOL
"Stanowisko_I2"	M 318.4	BOOL
"I2_Stan_Ma_Zadanie"	M 318.5	BOOL
"Edge_M318.6"	M 318.6	BOOL
"Help_318.7"	M 318.7	BOOL
"I3_Kier_Pob_Spedycja"	M 319.0	BOOL
"I3_Kier_Pob_Intro"	M 319.1	BOOL
"I3_Buff_Wiaz_Pop"	M 319.2	BOOL
"I3_Buff_Wiaz_Wzdl"	M 319.3	BOOL
"I3_Buff_Kod_0"	M 320.0	BOOL
"I3_Buff_Kod_1"	M 320.1	BOOL
"I3_Buff_Kod_2"	M 320.2	BOOL
"I3_Buff_Kod_3"	M 320.3	BOOL
"Stanowisko_I3"	M 320.4	BOOL
"I3_Stan_Ma_Zadanie"	M 320.5	BOOL
"Edge_M320.6"	M 320.6	BOOL
"Help_320.7"	M 320.7	BOOL
"Brak_komunikacj_Gender"	M 400.0	BOOL
"Wspolny_Auto"	M 401.0	BOOL
"Wspolny_Reczny"	M 401.1	BOOL
"Zbocze_M401.2"	M 401.2	BOOL
"Gender_Zalacz_Auto_Woz"	M 401.7	BOOL	// Gender ma zalaczyc auto wozkowi
"Gender_Auto_Reczny"	M 404.0	BOOL
"Reset_Read"	M 501.0	BOOL	// Przycisk resetu transmisji
"Toggle_Para"	M 501.1	BOOL
"BL_Read_K_KB1"	M 502.0	BOOL
"Bl_Na_Write_K_KB1"	M 502.1	BOOL
"Help_Timmer_KB"	M 502.2	BOOL
"Help_M502.3"	M 502.3	BOOL
"Kier_KB1_Koniec_Read"	M 502.5	BOOL
"Kier_KB1_Koniec_Send"	M 502.6	BOOL
"Aktywna_Funkcja_KB"	M 502.7	BOOL
"Bl_Na_Read_K_Rot"	M 503.0	BOOL
"Bl_Na_Write_K_Rot"	M 503.1	BOOL
"Help_Timmer_Rot"	M 503.2	BOOL
"Help_M503.3"	M 503.3	BOOL
"Kier_Rot_Koniec_Read"	M 503.5	BOOL
"Kier_Rot_Koniec_Send"	M 503.6	BOOL
"Aktywna_Funkcja_Rot"	M 503.7	BOOL
"Bl_Na_Read_Para"	M 504.0	BOOL
"Bl_Na_Write_Para"	M 504.1	BOOL
"Help_Timmer_Para"	M 504.2	BOOL
"Help_M504.3"	M 504.3	BOOL
"Para_Koniec_Read"	M 504.5	BOOL
"Para_Koniec_Send"	M 504.6	BOOL
"Aktywna_Funkcja_Para"	M 504.7	BOOL
"Bl_Na_Read_Odb"	M 505.0	BOOL
"Bl_Na_Write_Odb"	M 505.1	BOOL
"Help_Timmer_Odb"	M 505.2	BOOL
"Help_M505.3"	M 505.3	BOOL
"Odb_Koniec_Read"	M 505.5	BOOL
"Odb_Koniec_Send"	M 505.6	BOOL
"Aktywna_Funkcja_Odb"	M 505.7	BOOL
"Edge_M513.0"	M 513.0	BOOL
"Edge_M513.1"	M 513.1	BOOL
"Edge_513.4"	M 513.4	BOOL
"Edge_M513.5"	M 513.5	BOOL
"Edge_M514.0"	M 514.0	BOOL
"M514.1"	M 514.1	BOOL
"Edge_M514.3"	M 514.3	BOOL
"Edge_M514.4"	M 514.4	BOOL
"Edge_M523.0"	M 523.0	BOOL
"Edge_M523.1"	M 523.1	BOOL
"Edge_M533.0"	M 533.0	BOOL
"Edge_M533.1"	M 533.1	BOOL
"Paleta_Obecna_Na_KB1"	M 600.0	BOOL
"Paleta_Obecna_Na_KB2"	M 600.1	BOOL
"Paleta_Obecna_Pob_I1"	M 600.3	BOOL
"Paleta_Obecna_Pob_I2"	M 600.4	BOOL
"Paleta_Obecna_Pob_I3"	M 600.5	BOOL
"Foto_Pokryte_Czasowo"	M 600.6	BOOL
"Foto_Odkryte_Czasowo"	M 600.7	BOOL
"Wpisz_Wartosc_Do_Stosu"	M 601.0	BOOL
"Kasuj_Rekord_W_Kolejce"	M 601.1	BOOL
"Pobierz_Wartosc"	M 601.2	BOOL
"Potwierdzenie_Wpisania"	M 602.0	BOOL
"Potwierdzenie_Pobrania"	M 602.1	BOOL
"Potwierdzenie_Kasowania"	M 602.2	BOOL
"Help_M602.3"	M 602.3	BOOL
"Help_M602.4"	M 602.4	BOOL
"Help_M602.5"	M 602.5	BOOL
"Przejmij_Z_KB1"	M 603.0	BOOL
"Przejmij_Z_KB2"	M 603.1	BOOL
"Przejmij_Z_I1"	M 603.2	BOOL
"Oddaj_Na_Spedycje"	M 603.3	BOOL
"Oddaj_Na_Intro"	M 603.4	BOOL
"Przejmij_z_I2"	M 603.5	BOOL
"Przejmij_z_I3"	M 603.6	BOOL
"Wozek_Na_Reczny"	M 605.0	BOOL
"Wozek_Na_Auto"	M 605.1	BOOL
"Edge_M606.0"	M 606.0	BOOL
"Edge_M606.1"	M 606.1	BOOL
"Edge_M606.2"	M 606.2	BOOL
"Edge_M606.3"	M 606.3	BOOL
"KB1_Przej_Auto_Na_Recz"	M 607.0	BOOL
"KB2_Przej_Auto_Na_Recz"	M 607.1	BOOL
"Buff_Przejscie_Na_Recz"	M 607.2	BOOL
"Gen_Przejscie_Na_Reczny"	M 607.3	BOOL
"Edge_M608.0"	M 608.0	BOOL
"Edge_M608.1"	M 608.1	BOOL
"Edge_M608.2"	M 608.2	BOOL
"Edge_M608.3"	M 608.3	BOOL
"Warunk_Zasprz_KB1"	M 609.0	BOOL
"Warunk_Zasprz_KB2"	M 609.1	BOOL
"Warunk_Zasprz_Buffory"	M 609.2	BOOL
"Warunk_Zasprz_Gender"	M 609.3	BOOL
"Wozek_Kier_Spedycja"	M 610.0	BOOL
"Wozek_Kier_Intro"	M 610.1	BOOL
"Wozek_Info_Bit_0"	M 611.0	BOOL
"Wozek_Info_Bit_1"	M 611.1	BOOL
"Wozek_Info_Bit_2"	M 611.2	BOOL
"Wozek_Info_Bit_3"	M 611.3	BOOL
"Edge_M612.0"	M 612.0	BOOL
"Help_M612.1"	M 612.1	BOOL
"Paleta_Od_KB12"	M 615.0	BOOL
"Pozcja_Wozek_Zadana"	MD 10	DINT
"Offset_Pozycji"	MD 14	DINT
"Gorny_Zakres_Pozycji_Ok"	MD 28	DINT
"Dolny_Zakres_Pozycji_Ok"	MD 32	DINT
"KB1_MD140"	MD 140	DINT
"KB1_Cale_Zadanie"	MD 148	DWORD
"KB2_MD240"	MD 240	DINT
"KB2_Cale_Zadanie"	MD 248	DINT
"Help_MD340"	MD 340	DINT
"I1_Buff_Mask_Dword"	MD 360	DWORD
"I2_Buff_Mask_Dword"	MD 380	DWORD
"Help_MD382"	MD 382	DINT
"Help_MD384"	MD 384	DINT
"I3_Buff_Mask_Dword"	MD 390	DWORD
"I3_Help_MD394"	MD 394	DINT
"Wartosc_Dla_Wozka"	MD 620	DINT
"Wartosc_Wyjsciowa_Sortu"	MD 624	DINT
"Help_MD628"	MD 628	DWORD
"Kod_Przejdu_Do_Wozka"	MD 634	DINT
"War_KB1_Waga"	MD 650	DINT
"War_KB2_Waga"	MD 654	DINT
"War_I1_Waga"	MD 658	DINT
"War_I2_Waga"	MD 662	DINT
"War_I3_Waga"	MD 666	DINT
"Rejestr_Wozka"	MD 680	DWORD
"Wartosc_Bufforu_Help"	MD 720	DWORD
"KB1_Rozkaz_Zadania"	MW 148	WORD
"Wartosc_Bufforu_W_Kol"	MW 160	INT
"KB2_Rozkaz_Zadania"	MW 248	WORD
"Help_MW350"	MW 350	WORD
"Help_MW352"	MW 352	WORD
"Help_MW354"	MW 354	WORD
"Help_Mw356"	MW 356	WORD
"Help_MW358"	MW 358	WORD
"I1_Buff_Maska_Z_HMI"	MW 360	WORD
"Help_MW370"	MW 370	WORD
"Help_MW372"	MW 372	WORD
"Help_MW374"	MW 374	WORD
"Help_MW376"	MW 376	WORD
"Help_MW378"	MW 378	WORD
"I2_Buff_Maska_Z_HMI"	MW 380	WORD
"I3_Buff_Maska_Z_HMI"	MW 390	WORD
"I2_Help_MW412"	MW 412	WORD
"I2_Help_MW414"	MW 414	WORD
"I3_Help_MW416"	MW 416	WORD
"I3_Help_MW418"	MW 418	WORD
"Help_MW520"	MW 520	WORD
"Help_MW522"	MW 522	WORD
"Petla_Read_Kier_KB1"	MW 524	INT
"Petla_Send_Kier_KB1"	MW 526	INT
"MW530"	MW 530	WORD
"Help_MW532"	MW 532	WORD
"Petla_Read_Kier_Rot"	MW 534	INT
"Petla_Send_Kier_Rot"	MW 536	INT
"Help_MW540"	MW 540	WORD
"Help_MW542"	MW 542	WORD
"Petla_Read_Para"	MW 544	INT
"Petla_Send_Para"	MW 546	INT
"Help_MW628"	MW 628	WORD
"MW_Kolejka_KB1"	MW 670	INT
"MW_Kolejka_KB2"	MW 672	INT
"MW_Kolejka_I1"	MW 674	INT
"MW_Kolejka_I2"	MW 676	INT
"MW_Kolejka_I3"	MW 678	INT
"I/O_FLT1"	OB 82	OB 82	// I/O Point Fault 1
"RACK_FLT"	OB 86	OB 86	// Loss of Rack Fault
"COMM_FLT"	OB 87	OB 87	// Communication Fault
"PROG_ERR"	OB 121	OB 121	// Programming Error
"MOD_ERR"	OB 122	OB 122	// Module Access Error
"Buff_Lam_Przek_Bezp_O"	Q 8.0	BOOL	// Przekaznik bezpieczenstwa buffory ok
"Buff_Lampka_Pol_Auto"	Q 8.1	BOOL
"Buffor_Lampka_Auto"	Q 8.2	BOOL
"q_Buff_Zal_Wozka"	Q 8.3	BOOL
"q_Reset_P_Bezp_KB1"	Q 8.4	BOOL	// Reset przekaznika bezpieczenstwa Wozka KB1 s.18
"q_Reset_P_Bezp_KB2"	Q 8.5	BOOL	// Reset przekaznika bezpieczenstwa Wozka KB2 s.18
"Rezerwa_Q8.6"	Q 8.6	BOOL
"Rezerwa_Q8.7"	Q 8.7	BOOL
"Rezerwa_Q9.0"	Q 9.0	BOOL
"Rezerwa_Q9.1"	Q 9.1	BOOL
"Buff_Lampa_Kol_Buf_Ziel"	Q 9.2	BOOL
"Buff_Lampa_Kol_Buf_Pom"	Q 9.3	BOOL
"Buff_Lampa_Kol_Buf_Czer"	Q 9.4	BOOL
"Buff_Lampa_Kol_Buf_Nieb"	Q 9.5	BOOL
"Buff_Lampa_Kol_Buf_Syg"	Q 9.6	BOOL
"Rezerwa_Q9.7"	Q 9.7	BOOL
"Buff_Reset_Przek_Bezp"	Q 10.0	BOOL
"Buff_Reset_Przek_Bezp_1"	Q 10.1	BOOL
"Buff_Reset_Przeka_Bezp_2"	Q 10.2	BOOL
"Buff_Swiatlo_Zielone"	Q 10.3	BOOL	// Swiatlo zielone drogowe
"Buff_Swiatl_Czerwone"	Q 10.4	BOOL
"Rezerwa_Q10.5"	Q 10.5	BOOL
"Rezerwa_Q10.6"	Q 10.6	BOOL
"Rezerwa_Q10.7"	Q 10.7	BOOL
"Buff_Lampa_Kol_Gen_Ziel"	Q 11.0	BOOL	// S
"Buff_Lampa_Kol_Gen_Pom"	Q 11.1	BOOL	// str 21
"Buff_Lampa_Kol_Gen_Czer"	Q 11.2	BOOL	// str 21
"Buff_Lampa_Kol_Gen_Bial"	Q 11.3	BOOL	// str 21
"Buff_Lampa_Kol_Gen_Syg"	Q 11.4	BOOL	// str 21
"Rezerwa_Q11.6"	Q 11.5	BOOL	// str 21
"KB1_PB_Strefa_B_Lampka"	Q 12.0	BOOL	// Lapmka strefa bezpieczenstwa ok
"KB1_PB_Semi_Auto_Lampka"	Q 12.1	BOOL	// Lampka polautomatyka
"KB1_PB_Auto_Lampka"	Q 12.2	BOOL	// Lampka auto
"KB1_PB_Funkcja_Lampka"	Q 12.3	BOOL	// Lampka przycisku funkcyjnego
"KB1_PB_B_Winda_Lampka"	Q 12.4	BOOL	// Lampka piorka winda
"KB1_PB_B_Obr_Lampka"	Q 12.5	BOOL	// Lampka piorka obrotnica
"KB1_Rezerwa_Q22.6"	Q 12.6	BOOL
"KB1_Rezerwa_Q22.7"	Q 12.7	BOOL
"KB1_Lampa_Wyb_Kier_Lewo"	Q 13.0	BOOL
"KB1_Lampa_Wyb_Kier_Prawo"	Q 13.1	BOOL
"KB1_Lampa_Kol_Ziel"	Q 13.2	BOOL	// Lampka kolor zielony str 19
"KB1_Lampa_Kol_Pom"	Q 13.3	BOOL	// Lampka kolor pomaranczowy str 19
"KB1_Lampa_Kol_Czerw"	Q 13.4	BOOL	// Lampka kolor czerwony str 19
"KB1_Lampa_Kol_Nieb"	Q 13.5	BOOL
"KB1_Syrena"	Q 13.6	BOOL
"KB1_Lampa_Blysk_Wozek"	Q 13.7	BOOL
"KB1_Winda_Silnik_Pompa"	Q 14.0	BOOL
"KB1_Winda_Zawor"	Q 14.1	BOOL
"KB1_Reset_Przek_Bezp"	Q 14.2	BOOL
"KB1_Odblokuj_Lenze"	Q 14.3	BOOL
"KB1_Przek_Rez_K20.5"	Q 14.4	BOOL
"KB1_Odblokuj_Ham_Sew"	Q 14.5	BOOL
"KB1_Odblokuj_Ham_Lenze"	Q 14.6	BOOL
"KB1_Rezerwa_Q24.7"	Q 14.7	BOOL
"KB1_Fal_Seg_Przod"	Q 15.0	BOOL
"KB1_Fal_Segbert_Tyl"	Q 15.1	BOOL
"KB2_PB_Strefa_B_Lampka"	Q 22.0	BOOL	// Lapmka strefa bezpieczenstwa ok
"KB2_PB_Semi_Auto_Lampka"	Q 22.1	BOOL	// Lampka polautomatyka
"KB2_PB_Auto_Lampka"	Q 22.2	BOOL	// Lampka auto
"KB2_PB_Funkcja_Lampka"	Q 22.3	BOOL	// Lampka przycisku funkcyjnego
"KB2_PB_B_Winda_Lampka"	Q 22.4	BOOL	// Lampka piorka winda
"KB2_PB_B_Obr_Lampka"	Q 22.5	BOOL	// Lampka piorka obrotnica
"KB2_Rezerwa_Q22.6"	Q 22.6	BOOL
"KB2_Rezerwa_Q22.7"	Q 22.7	BOOL
"KB2_Lampa_Wyb_Kier_Lewo"	Q 23.0	BOOL
"KB2_Lampa_Wyb_Kier_Prawo"	Q 23.1	BOOL
"KB2_Lampa_Kol_Ziel"	Q 23.2	BOOL	// Lampka kolor zielony str 19
"KB2_Lampa_Kol_Pom"	Q 23.3	BOOL	// Lampka kolor pomaranczowy str 19
"KB2_Lampa_Kol_Czerw"	Q 23.4	BOOL	// Lampka kolor czerwony str 19
"KB2_Lampa_Kol_Nieb"	Q 23.5	BOOL
"KB2_Syrena"	Q 23.6	BOOL
"KB2_Lampa_Blysk_Wozek"	Q 23.7	BOOL
"KB2_Winda_Silnik_Pompa"	Q 24.0	BOOL
"KB2_Winda_Zawor"	Q 24.1	BOOL
"KB2_Reset_Przek_Bezp"	Q 24.2	BOOL
"KB2_Odblokuj_Lenze"	Q 24.3	BOOL
"KB2_Przek_Rez_K20.5"	Q 24.4	BOOL
"KB2_Odblokuj_Ham_Sew"	Q 24.5	BOOL
"KB2_Odblokuj_Ham_Lenze"	Q 24.6	BOOL
"KB2_Rezerwa_Q24.7"	Q 24.7	BOOL
"KB2_Fal_Seg_Przod"	Q 25.0	BOOL
"KB2_Fal_Seg_Tyl"	Q 25.1	BOOL
"op_Bit_Komunikacji"	Q 38.0	BOOL	// Bit komunikacji do Shuttle(-->Shuttle)
"op_Bit_Nowej_Pozycji"	Q 39.1	BOOL	// Bit zadania nowej pozycji (-->Shuttle)
"op_Potw_Pozycji"	Q 39.2	BOOL	// Bit potwierdzenia pzosycji (-->Shuttle)
"op_Bit_Rezerwy_38_3"	Q 39.3	BOOL	// Bit rezerwy 38.3
"op_Zasprz_Wozka"	Q 39.4	BOOL	// Rozkaz Zasprzeglenie Wozka (-->Shuttle)
"op_Rozprz_Wozka"	Q 39.5	BOOL	// Rozkaz Rozprzeglenie Wozka (--> Shuttle)
"op_Silnik_Banda_Lewo"	Q 39.6	BOOL	// Jazda silnika w lewo (-->Shuttle)
"op_Silnik_Banda_Prawo"	Q 39.7	BOOL	// Jazda silnika w prawo
"Buff_1_Wlot_1_Wiaz_Pop"	Q 80.0	BOOL
"Buff_1_Wlot_1_Wiaz_Wzdl"	Q 80.1	BOOL
"Buff_1_Wlot_1_Dekl"	Q 80.2	BOOL
"Buff_1_Wlot_1_Fol"	Q 80.3	BOOL
"Buff_2_Wlot_2_Wiaz_Pop"	Q 80.4	BOOL
"Buff_2_Wlot_2_Wiaz_Wzdl"	Q 80.5	BOOL
"Buff_2_Wlot_2_Dekl"	Q 80.6	BOOL
"Buff_2_Wlot_2_Fol"	Q 80.7	BOOL
"Buff_2_Wlot_3_Wiaz_Pop"	Q 81.0	BOOL
"Buff_2_Wlot_3_Wiaz_Wzdl"	Q 81.1	BOOL
"Buff_2_Wlot_3_Dekl"	Q 81.2	BOOL
"Buff_2_Wlot_3_Fol"	Q 81.3	BOOL
"Buff_2_Lampka_Strefa_B"	Q 82.0	BOOL
"Buff_2_Lampka_Pol_Auto"	Q 82.1	BOOL
"Buff_2_Lampka_Auto"	Q 82.2	BOOL
"DWORD_8_Shuttle"	QD 38	DWORD
"QD42_Pozycja_Zadana"	QD 42	DINT	// Pozycja zadana w mm (--> Shuttle)
"READ_CLK"	SFC 1	SFC 1	// Read System Clock
"DPNRM_DG"	SFC 13	SFC 13	// Read Diagnostic Data of a DP Slave
"DPRD_DAT"	SFC 14	SFC 14	// Read Consistent Data of a Standard DP Slave
"DPWR_DAT"	SFC 15	SFC 15	// Write Consistent Data to a Standard DP Slave
"BLKMOV"	SFC 20	SFC 20	// Copy Variables
"READ_ERR"	SFC 38	SFC 38	// Read Error Registers
"WR_REC"	SFC 58	SFC 58	// Write Data Record
"RD_REC"	SFC 59	SFC 59	// Read a Data Record
"Timer_0_Czerwone"	T 0	TIMER
"Timer_T1"	T 1	TIMER
"Shuttle_T2"	T 2	TIMER
"Help_T4"	T 4	TIMER
"KB1_T10"	T 10	TIMER
"KB1_T11"	T 11	TIMER
"KB1_T12"	T 12	TIMER
"KB1_T13"	T 13	TIMER
"KB1_T14"	T 14	TIMER
"KB1_T15"	T 15	TIMER
"KB1_Opoznienie_Startu"	T 16	TIMER
"KB1_Filtr_Segbert"	T 17	TIMER
"KB1_T18"	T 18	TIMER
"T19"	T 19	TIMER
"KB2_T20"	T 20	TIMER
"KB2_T21"	T 21	TIMER
"KB2_T22"	T 22	TIMER
"KB2_T23"	T 23	TIMER
"KB2_T24"	T 24	TIMER
"KB2_T25"	T 25	TIMER
"KB2_Opoznienie_Startu"	T 26	TIMER
"KB2_Filtr_Segbert"	T 27	TIMER
"KB2_T28"	T 28	TIMER
"T29"	T 29	TIMER
"200ms_T31"	T 31	TIMER
"500ms_T32"	T 32	TIMER
"100ms_T33"	T 33	TIMER
"Buff_T35"	T 35	TIMER
"Buff_T36"	T 36	TIMER
"Buff_T37"	T 37	TIMER
"Kontrola_T40"	T 40	TIMER
"Kontrola_T41"	T 41	TIMER
"Kontrola_T42"	T 42	TIMER
"Kontrola_T43"	T 43	TIMER
"Kontrola_T44"	T 44	TIMER
"Kontrola_T45"	T 45	TIMER
"Kontrola_T46"	T 46	TIMER
"Kontrola_T47"	T 47	TIMER
"Kontrola_T48"	T 48	TIMER
"Kontrola_T49"	T 49	TIMER
"KB1_T50"	T 50	TIMER
"KB1_T51"	T 51	TIMER
"KB1_T52"	T 52	TIMER
"Kontrola_T53"	T 53	TIMER
"Kontrola_T54"	T 54	TIMER
"Kontrola_T55"	T 55	TIMER
"Kontrola_T56"	T 56	TIMER
"KB2_T60"	T 60	TIMER
"KB2_T61"	T 61	TIMER
"KB2_T62"	T 62	TIMER
"BUF_T70"	T 70	TIMER
"T71_Opoznienie_Rozp"	T 71	TIMER
"Timer_Wozek_Pokryte"	T 72	TIMER
"Timer_Wozek_Odkryte"	T 73	TIMER
"T75"	T 75	TIMER
"T76"	T 76	TIMER
"T77"	T 77	TIMER
"T78"	T 78	TIMER
"T79"	T 79	TIMER
"Help_T80"	T 80	TIMER
"Help_T81"	T 81	TIMER
"Help_T82"	T 82	TIMER
"Help_T90"	T 90	TIMER
"KB2_Timer_Winda_91"	T 91	TIMER
"KB2_Timer_Winda_92"	T 92	TIMER
"KB1_Timer_Winda_93"	T 93	TIMER
"KB1_Timer_Winda_94"	T 94	TIMER
"T100"	T 100	TIMER
"T_100_Wozek_Na_Auto"	T 101	TIMER
"Timmer_102_KB1"	T 102	TIMER
"Timer_103_KB2"	T 103	TIMER
"Timmer_104_Pobieranie"	T 104	TIMER
"Timmer_105_Odbieranie"	T 105	TIMER
"Help_T107"	T 107	TIMER
"Help_T108"	T 108	TIMER
"T109"	T 109	TIMER
"Timmer_T110"	T 110	TIMER
"Timmer_T111"	T 111	TIMER
"Timmer_Pob_I2"	T 112	TIMER
"Timmer_Pob_I3"	T 113	TIMER
"Timer_T120"	T 120	TIMER
"Help_T121"	T 121	TIMER
"T130"	T 130	TIMER
"T131"	T 131	TIMER
"T140"	T 140	TIMER
"T141"	T 141	TIMER
"TASMA_MODEL"	UDT 1	UDT 1	// Model Tasmy z Sew'em
"ESTOP_MODEL"	UDT 3	UDT 3
"OBROTNICA_MODEL"	UDT 6	UDT 6	// Model sygnalow z bandy obrotowej
"CZUJNIKI_MODEL_1"	UDT 7	UDT 7	// Model czujnikow na obrotnicy
"VAT_1"	VAT 1	
"Wejscia_Wysjcia"	VAT 2	
"VAT_DB701"	VAT 3	
"VAT_DB702"	VAT 4	
"VAT_kb2"	VAT 5	
"para"	VAT 6	
"VAT_Buffory"	VAT 7	
"VAT_Cargo"	VAT 8	
"buffory_2"	VAT 9	
END_SYMBOL_TABLE

FUNCTION "Wozek_Queue_V3" : VOID	// FC 408
AUTHOR : Kng
NAME : Fahren
VERSION : 0.1
VAR_INPUT
  _Paleta_KB1 : BOOL ;
  Kier_KB1_Gender : BOOL ;
  Kier_KB1_Intro : BOOL ;
  Wartosc_KB1 : INT ;
  Kod_KB1 : BYTE ;
  _Paleta_KB2 : BOOL ;
  Kier_KB2_Gender : BOOL ;
  Kier_KB2_Intro : BOOL ;
  Wartosc_KB2 : INT ;
  Kod_KB2 : BYTE ;
  _Paleta_I1 : BOOL ;	//Intro pobieranie nr 1
  Kier_I1_Gender : BOOL ;
  Kier_I1_Intro : BOOL ;
  Wartosc_I1 : INT ;
  Kod_I1 : BYTE ;
  _Paleta_I2 : BOOL ;	//Intro pobieranie nr 2
  Kier_I2_Gender : BOOL ;
  Kier_I2_Intro : BOOL ;
  Wartosc_I2 : INT ;
  Kod_I2 : BYTE ;
  _Paleta_I3 : BOOL ;	//Intro pobieranie nr 2
  Kier_I3_Gender : BOOL ;
  Kier_I3_Intro : BOOL ;
  Wartosc_I3 : INT ;
  Kod_I3 : BYTE ;
END_VAR
VAR_OUTPUT
  od_Wartosc_KB1 : DINT ;
  od_Wartosc_KB2 : DINT ;
  od_Wartosc_I1 : DINT ;
  od_Wartosc_I2 : DINT ;
  od_Wartosc_I3 : DINT ;
END_VAR
VAR_TEMP
  Slowo_LW0 : INT ;
  Slowo_LW2 : INT ;
  Temp_Help_1 : BOOL ;
END_VAR
BEGIN
NETWORK
TITLE =
//Ten Network celowo jest wolny
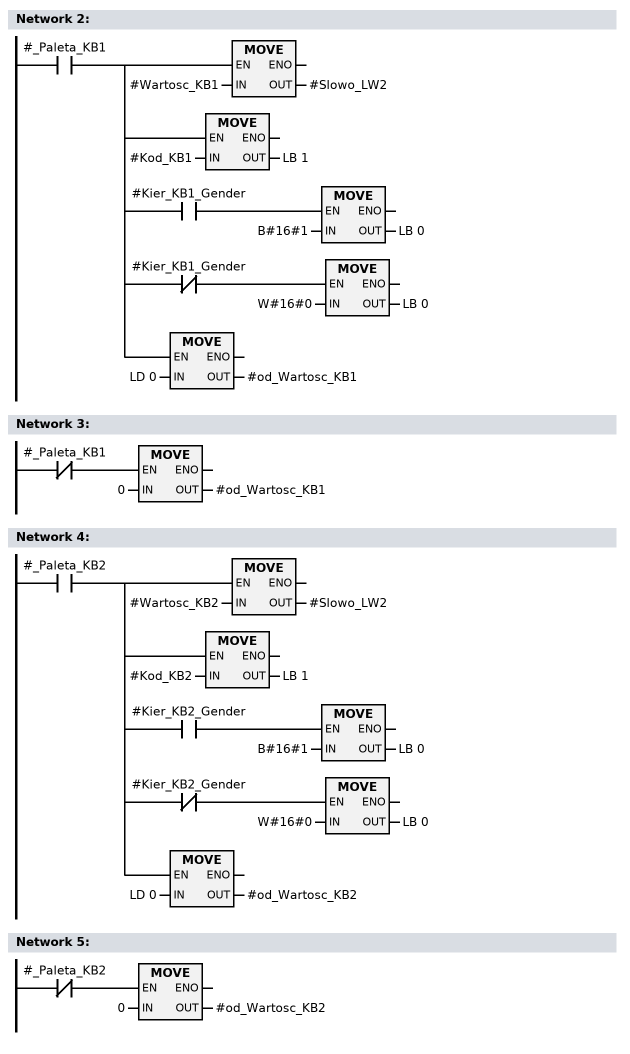
NETWORK
TITLE =
//Budowanie wartosci transferowej :
//LB0-kierunek intro(1),spedycja(0)
//LB1-Kod maszyny np KB1-1
//LW2-Wartosc wagowa
      A     #_Paleta_KB1;
      =     L 5.0;
      A     L 5.0;
      JNB   _001;
      L     #Wartosc_KB1;
      T     #Slowo_LW2;
_001: NOP   0;
      A     L 5.0;
      JNB   _002;
      L     #Kod_KB1;
      T     LB 1;
_002: NOP   0;
      A     L 5.0;
      A     #Kier_KB1_Gender;
      JNB   _003;
      L     B#16#1;
      T     LB 0;
_003: NOP   0;
      A     L 5.0;
      AN    #Kier_KB1_Gender;
      JNB   _004;
      L     W#16#0;
      T     LB 0;
_004: NOP   0;
      A     L 5.0;
      JNB   _005;
      L     LD 0;
      T     #od_Wartosc_KB1;
_005: NOP   0;
NETWORK
TITLE =
      AN    #_Paleta_KB1;
      JNB   _006;
      L     0;
      T     #od_Wartosc_KB1;
_006: NOP   0;
NETWORK
TITLE =
//Budowanie wartosci transferowej dla kb2
      A     #_Paleta_KB2;
      =     L 5.0;
      A     L 5.0;
      JNB   _007;
      L     #Wartosc_KB2;
      T     #Slowo_LW2;
_007: NOP   0;
      A     L 5.0;
      JNB   _008;
      L     #Kod_KB2;
      T     LB 1;
_008: NOP   0;
      A     L 5.0;
      A     #Kier_KB2_Gender;
      JNB   _009;
      L     B#16#1;
      T     LB 0;
_009: NOP   0;
      A     L 5.0;
      AN    #Kier_KB2_Gender;
      JNB   _00a;
      L     W#16#0;
      T     LB 0;
_00a: NOP   0;
      A     L 5.0;
      JNB   _00b;
      L     LD 0;
      T     #od_Wartosc_KB2;
_00b: NOP   0;
NETWORK
TITLE =
//jezeli brak palety na kb2 to przypisz 0
      AN    #_Paleta_KB2;
      JNB   _00c;
      L     0;
      T     #od_Wartosc_KB2;
_00c: NOP   0;
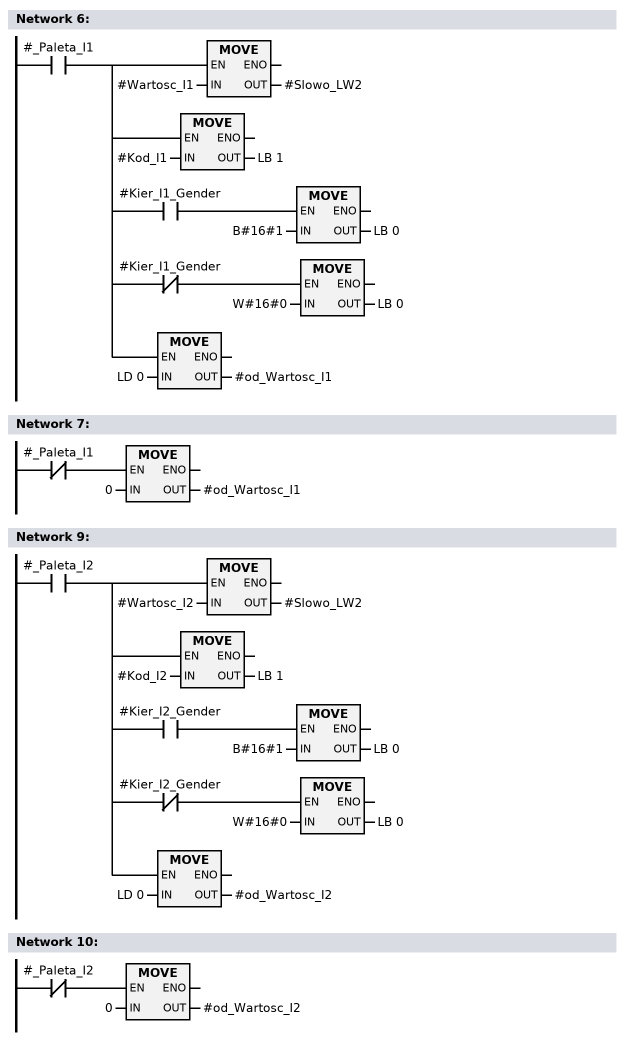
NETWORK
TITLE =
//Budowanie wartosci transferowej dla intro
      A     #_Paleta_I1;
      =     L 5.0;
      A     L 5.0;
      JNB   _00d;
      L     #Wartosc_I1;
      T     #Slowo_LW2;
_00d: NOP   0;
      A     L 5.0;
      JNB   _00e;
      L     #Kod_I1;
      T     LB 1;
_00e: NOP   0;
      A     L 5.0;
      A     #Kier_I1_Gender;
      JNB   _00f;
      L     B#16#1;
      T     LB 0;
_00f: NOP   0;
      A     L 5.0;
      AN    #Kier_I1_Gender;
      JNB   _010;
      L     W#16#0;
      T     LB 0;
_010: NOP   0;
      A     L 5.0;
      JNB   _011;
      L     LD 0;
      T     #od_Wartosc_I1;
_011: NOP   0;
NETWORK
TITLE =
      AN    #_Paleta_I1;
      JNB   _012;
      L     0;
      T     #od_Wartosc_I1;
_012: NOP   0;
NETWORK
TITLE =
NETWORK
TITLE =
//Budowanie wartosci transferowej dla intro
      A     #_Paleta_I2;
      =     L 5.0;
      A     L 5.0;
      JNB   _013;
      L     #Wartosc_I2;
      T     #Slowo_LW2;
_013: NOP   0;
      A     L 5.0;
      JNB   _014;
      L     #Kod_I2;
      T     LB 1;
_014: NOP   0;
      A     L 5.0;
      A     #Kier_I2_Gender;
      JNB   _015;
      L     B#16#1;
      T     LB 0;
_015: NOP   0;
      A     L 5.0;
      AN    #Kier_I2_Gender;
      JNB   _016;
      L     W#16#0;
      T     LB 0;
_016: NOP   0;
      A     L 5.0;
      JNB   _017;
      L     LD 0;
      T     #od_Wartosc_I2;
_017: NOP   0;
NETWORK
TITLE =
//Kasuj buffor dla I2
      AN    #_Paleta_I2;
      JNB   _018;
      L     0;
      T     #od_Wartosc_I2;
_018: NOP   0;
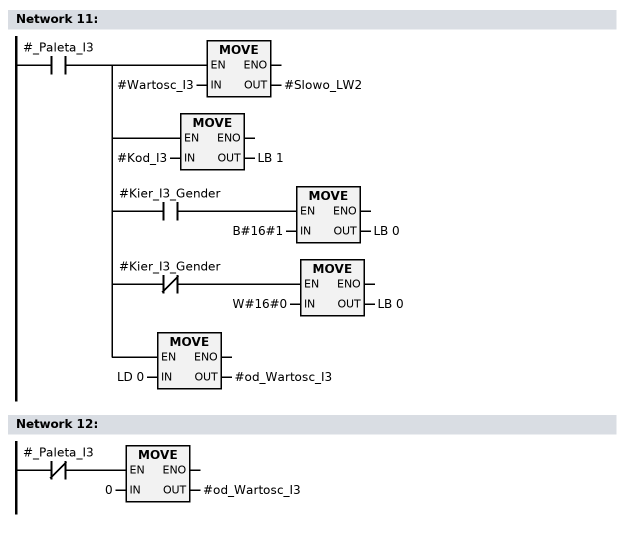
NETWORK
TITLE =
//Budowanie wartosci transferowej dla intro
      A     #_Paleta_I3;
      =     L 5.0;
      A     L 5.0;
      JNB   _019;
      L     #Wartosc_I3;
      T     #Slowo_LW2;
_019: NOP   0;
      A     L 5.0;
      JNB   _01a;
      L     #Kod_I3;
      T     LB 1;
_01a: NOP   0;
      A     L 5.0;
      A     #Kier_I3_Gender;
      JNB   _01b;
      L     B#16#1;
      T     LB 0;
_01b: NOP   0;
      A     L 5.0;
      AN    #Kier_I3_Gender;
      JNB   _01c;
      L     W#16#0;
      T     LB 0;
_01c: NOP   0;
      A     L 5.0;
      JNB   _01d;
      L     LD 0;
      T     #od_Wartosc_I3;
_01d: NOP   0;
NETWORK
TITLE =
//Kasuj buffor dla I2
      AN    #_Paleta_I3;
      JNB   _01e;
      L     0;
      T     #od_Wartosc_I3;
_01e: NOP   0;
END_FUNCTION

FUNCTION "Sorting_V3" : VOID	// FC 409
//Funkcja odpowiada za sortowanie elementow dostarczonych do bloku db. Sortowanie 
//odbywa sie automatcycznie. Wpisanie nastepuje przez zbocze na wejsciu wpisz 
//wartosc.
//
//Funkcja odnosi sie bezposrednio do bloku danych db402
//
//
//
//
AUTHOR : Kng
NAME : Help_FC
VERSION : 0.1
VAR_INPUT
  id_Wartosc_KB1 : DINT ;	//Wpisuje nowy rekord na dol bloku
  id_Wartosc_KB2 : DINT ;	//Pobiera rekord z gory bloku
  id_Wartosc_I1 : DINT ;	//Kasuje rekord od wartosci wsadowej
  id_Wartosc_I2 : DINT ;
  id_Wartosc_I3 : DINT ;
  i_Poz_5_Down : BOOL ;
  i_Poz_4_Up : BOOL ;
  i_Poz_4_Down : BOOL ;
  i_Poz_3_Up : BOOL ;
  i_Poz_3_Down : BOOL ;
  i_Poz_2_Up : BOOL ;
  i_Poz_2_Down : BOOL ;
  i_Poz_1_Up : BOOL ;
END_VAR
VAR_IN_OUT
  iow_Help_DWord : DWORD ;
END_VAR
VAR_TEMP
  P : STRUCT
   KB1_Wpis : BOOL ;
   KB2_Wpis : BOOL ;
   I1_Wpis : BOOL ;
   I2_Wpis : BOOL ;
   I3_Wpis : BOOL ;
   KB1_Istnieje : BOOL ;
   KB2_Istnieje : BOOL ;
   I1_Istnieje : BOOL ;
   I2_Istnieje : BOOL ;
   I3_Istnieje : BOOL ;
   Help_Bit_0_7 : BOOL ;
   Wpis_0_istnieje : BOOL ;
   Wpis_1_istnieje : BOOL ;
   Wpis_2_istnieje : BOOL ;
   Wpis_3_istnieje : BOOL ;
   Wpis_4_istnieje : BOOL ;
   Wpis_5_istnieje : BOOL ;
   Wpis_6_istnieje : BOOL ;
   edge_1 : BOOL ;
   edge_2 : BOOL ;
   edge_3 : BOOL ;
   edge_4 : BOOL ;
   edge_5 : BOOL ;
   edge_6 : BOOL ;
  END_STRUCT ;
  Help_Blok_Move : INT ;
  Help_Int_2 : INT ;
  Help_Dint : DINT ;
  Wpis : STRUCT
   _0_dbb0_Kod_Kier : BYTE ;
   _0_dbb1_Kod_Maszyna : BYTE ;
   _0_dbw2_War_Wagowa : INT ;
   _1_dbb4_Kod_Kier : BYTE ;
   _1_dbb5_Kod_Maszyna : BYTE ;
   _1_dbw6_War_Wagowa : INT ;
   _2_dbb8_Kod_Kier : BYTE ;
   _2_dbb9_Kod_Maszyna : BYTE ;
   _2_dbw10_War_Wagowa : INT ;
   _3_dbb12_Kod_Kier : BYTE ;
   _3_dbb13_Kod_Maszyna : BYTE ;
   _3_dbw14_War_Wagowa : INT ;
   _4_dbb16_Kod_Kier : BYTE ;
   _4_dbb17_Kod_Maszyna : BYTE ;
   _4_dbw18_War_Wagowa : INT ;
   _5_dbb20_Kod_Kier : BYTE ;
   _5_dbb21_Kod_Masz : BYTE ;
   _5_dbw22_War_Wagowa : INT ;
   _6_dbb24_Kod_Kier : BYTE ;
   _6_dbb25_Kod_Masz : BYTE ;
   _6_dbw26_War_Wagowa : INT ;
   Kod_Spr_KB1 : BYTE ;
   Kod_Spr_KB2 : BYTE ;
   Kod_Spr_I1 : BYTE ;
   Kod_Spr_I2 : BYTE ;
   Kod_Spr_I3 : BYTE ;
   Kod_Spr_Rezerwa : BYTE ;
  END_STRUCT ;
  Temp_Wpis_KB1 : BOOL ;
  Temp_Wpis_KB2 : BOOL ;
  Temp_Wpis_I1 : BOOL ;
  Temp_Wpis_I2 : BOOL ;
  Temp_Wpis_I3 : BOOL ;
END_VAR
BEGIN
NETWORK
TITLE =
//Ten Network celowo jest wolny
NETWORK
TITLE =
//Zaladowanie bitow przejsciowych
      L     #iow_Help_DWord;
      T     #P;
//Zaladowanie pakietu danych
      CALL  "BLKMOV" (
           SRCBLK                   := "Key_DB".Wpis,
           RET_VAL                  := #Help_Blok_Move,
           DSTBLK                   := #Wpis);
NETWORK
TITLE =
//Sprawdz istniejacy wpis
      L     #id_Wartosc_KB1;
      L     0;
      <>D;
      =     #P.KB1_Istnieje;
      NOT;
      R     #P.KB1_Wpis;
//---
      L     #id_Wartosc_KB2;
      L     0;
      <>D;
      =     #P.KB2_Istnieje;
      NOT;
      R     #P.KB2_Wpis;
//---
      L     #id_Wartosc_I1;
      L     0;
      <>D;
      =     #P.I1_Istnieje;
      NOT;
      R     #P.I1_Wpis;
//---
      L     #id_Wartosc_I2;
      L     0;
      <>D;
      =     #P.I2_Istnieje;
      NOT;
      R     #P.I2_Wpis;
//---
      L     #id_Wartosc_I3;
      L     0;
      <>D;
      =     #P.I3_Istnieje;
      NOT;
      R     #P.I3_Wpis;
NETWORK
TITLE =
//Zaladuj kody maszyn do sprawdzenia
//****KB1*************************************
      L     #id_Wartosc_KB1;
      T     #Help_Dint;
//Zaladuj bit odpowiedzialny za maszyne (kod maszyny)
      L     LB 9;
      T     #Wpis.Kod_Spr_KB1;
//****KB2*************************************
      L     #id_Wartosc_KB2;
      T     #Help_Dint;
//Zaladuj bit odpowiedzialny za maszyne (kod maszyny)
      L     LB 9;
      T     #Wpis.Kod_Spr_KB2;
//****I1**************************************
      L     #id_Wartosc_I1;
      T     #Help_Dint;
//Zaladuj bit odpowiedzialny za maszyne (kod maszyny)
      L     LB 9;
      T     #Wpis.Kod_Spr_I1;
//****I2**************************************
      L     #id_Wartosc_I2;
      T     #Help_Dint;
//Zaladuj bit odpowiedzialny za maszyne (kod maszyny)
      L     LB 9;
      T     #Wpis.Kod_Spr_I2;
//****I3**************************************
      L     #id_Wartosc_I3;
      T     #Help_Dint;
//Zaladuj bit odpowiedzialny za maszyne (kod maszyny)
      L     LB 9;
      T     #Wpis.Kod_Spr_I3;
//Przeprowadzeni sprwdzenia   dbd 0
      O(;
      L     #Wpis._0_dbb1_Kod_Maszyna;
      L     #Wpis.Kod_Spr_KB1;
      ==I;
      );
      O(;
      L     #Wpis._0_dbb1_Kod_Maszyna;
      L     #Wpis.Kod_Spr_KB2;
      ==I;
      );
      O(;
      L     #Wpis._0_dbb1_Kod_Maszyna;
      L     #Wpis.Kod_Spr_I1;
      ==I;
      );
      O(;
      L     #Wpis._0_dbb1_Kod_Maszyna;
      L     #Wpis.Kod_Spr_I2;
      ==I;
      );
      O(;
      L     #Wpis._0_dbb1_Kod_Maszyna;
      L     #Wpis.Kod_Spr_I3;
      ==I;
      );
      JC    dbd0;
      L     0;
      T     #Wpis._0_dbb0_Kod_Kier;
      T     #Wpis._0_dbb1_Kod_Maszyna;
      T     #Wpis._0_dbw2_War_Wagowa;
dbd0: NOP   0;
//Przeprowadzeni sprwdzenia   dbd 4 (pozycja 2)
      O(;
      L     #Wpis._1_dbb5_Kod_Maszyna;
      L     #Wpis.Kod_Spr_KB1;
      ==I;
      );
      O(;
      L     #Wpis._1_dbb5_Kod_Maszyna;
      L     #Wpis.Kod_Spr_KB2;
      ==I;
      );
      O(;
      L     #Wpis._1_dbb5_Kod_Maszyna;
      L     #Wpis.Kod_Spr_I1;
      ==I;
      );
      O(;
      L     #Wpis._1_dbb5_Kod_Maszyna;
      L     #Wpis.Kod_Spr_I2;
      ==I;
      );
      O(;
      L     #Wpis._1_dbb5_Kod_Maszyna;
      L     #Wpis.Kod_Spr_I3;
      ==I;
      );
      JC    dbd4;
      L     0;
      T     #Wpis._1_dbb4_Kod_Kier;
      T     #Wpis._1_dbb5_Kod_Maszyna;
      T     #Wpis._1_dbw6_War_Wagowa;
dbd4: NOP   0;
//Przeprowadzeni sprwdzenia   dbd 8 (pozycja 3)
      O(;
      L     #Wpis._2_dbb9_Kod_Maszyna;
      L     #Wpis.Kod_Spr_KB1;
      ==I;
      );
      O(;
      L     #Wpis._2_dbb9_Kod_Maszyna;
      L     #Wpis.Kod_Spr_KB2;
      ==I;
      );
      O(;
      L     #Wpis._2_dbb9_Kod_Maszyna;
      L     #Wpis.Kod_Spr_I1;
      ==I;
      );
      O(;
      L     #Wpis._2_dbb9_Kod_Maszyna;
      L     #Wpis.Kod_Spr_I2;
      ==I;
      );
      O(;
      L     #Wpis._2_dbb9_Kod_Maszyna;
      L     #Wpis.Kod_Spr_I3;
      ==I;
      );
      JC    dbd8;
      L     0;
      T     #Wpis._2_dbb8_Kod_Kier;
      T     #Wpis._2_dbb9_Kod_Maszyna;
      T     #Wpis._2_dbw10_War_Wagowa;
dbd8: NOP   0;
//Przeprowadzeni sprwdzenia   dbd 12 (pozycja 4)
      O(;
      L     #Wpis._3_dbb13_Kod_Maszyna;
      L     #Wpis.Kod_Spr_KB1;
      ==I;
      );
      O(;
      L     #Wpis._3_dbb13_Kod_Maszyna;
      L     #Wpis.Kod_Spr_KB2;
      ==I;
      );
      O(;
      L     #Wpis._3_dbb13_Kod_Maszyna;
      L     #Wpis.Kod_Spr_I1;
      ==I;
      );
      O(;
      L     #Wpis._3_dbb13_Kod_Maszyna;
      L     #Wpis.Kod_Spr_I2;
      ==I;
      );
      O(;
      L     #Wpis._3_dbb13_Kod_Maszyna;
      L     #Wpis.Kod_Spr_I3;
      ==I;
      );
      JC    d_12;
      L     0;
      T     #Wpis._3_dbb12_Kod_Kier;
      T     #Wpis._3_dbb13_Kod_Maszyna;
      T     #Wpis._3_dbw14_War_Wagowa;
d_12: NOP   0;
//Przeprowadzeni sprwdzenia   dbd 16 (pozycja 5)
      O(;
      L     #Wpis._4_dbb17_Kod_Maszyna;
      L     #Wpis.Kod_Spr_KB1;
      ==I;
      );
      O(;
      L     #Wpis._4_dbb17_Kod_Maszyna;
      L     #Wpis.Kod_Spr_KB2;
      ==I;
      );
      O(;
      L     #Wpis._4_dbb17_Kod_Maszyna;
      L     #Wpis.Kod_Spr_I1;
      ==I;
      );
      O(;
      L     #Wpis._4_dbb17_Kod_Maszyna;
      L     #Wpis.Kod_Spr_I2;
      ==I;
      );
      O(;
      L     #Wpis._4_dbb17_Kod_Maszyna;
      L     #Wpis.Kod_Spr_I3;
      ==I;
      );
      JC    d_16;
      L     0;
      T     #Wpis._4_dbb16_Kod_Kier;
      T     #Wpis._4_dbb17_Kod_Maszyna;
      T     #Wpis._4_dbw18_War_Wagowa;
d_16: NOP   0;
NETWORK
TITLE =
//Kasowanie zer w rejestrze. Polega na przesuwaniu wszystkiego w gore i tym samym 
//luki sa wycinane.Gdy zniknie paleta stos wycina element i przsuwa reszte w 
//gore.
//**********Pozycja 12.0
      L     LD 12;
      L     0;
      ==D;
      JCN   o1;
      L     LD 16;
      T     LD 12;
      L     LD 20;
      T     LD 16;
      L     LD 24;
      T     LD 20;
      L     LD 28;
      T     LD 24;
      L     LD 32;
      T     LD 28;
o1:   NOP   0;
//**********Pozycja 16.0
      L     LD 16;
      L     0;
      ==D;
      JCN   o2;
      L     LD 20;
      T     LD 16;
      L     LD 24;
      T     LD 20;
      L     LD 28;
      T     LD 24;
      L     LD 32;
      T     LD 28;
o2:   NOP   0;
//**********Pozycja 20.0
      L     LD 20;
      L     0;
      ==D;
      JCN   o3;
      L     LD 24;
      T     LD 20;
      L     LD 28;
      T     LD 24;
      L     LD 32;
      T     LD 28;
o3:   NOP   0;
//**********Pozycja 24.0
      L     LD 24;
      L     0;
      ==D;
      JCN   o4;
      L     LD 28;
      T     LD 24;
      L     LD 32;
      T     LD 28;
o4:   NOP   0;
//**********Pozycja 28.0
      L     LD 28;
      L     0;
      ==D;
      JCN   o5;
      L     LD 32;
      T     LD 28;
o5:   NOP   0;
NETWORK
TITLE =
//Zaladowanie nowej wartosci do KB1
//Wyresetuj bity tymczasowe
      SET;
      R     #Temp_Wpis_KB1;
      R     #Temp_Wpis_KB2;
      R     #Temp_Wpis_I1;
      R     #Temp_Wpis_I2;
      R     #Temp_Wpis_I3;
      A     #P.KB1_Istnieje;
      AN    #P.KB1_Wpis;
      JCN   z0;
      L     #id_Wartosc_KB1;
      T     #Help_Dint;
      AN    #P.KB1_Wpis;
      =     #Temp_Wpis_KB1;
      JU    x0;
z0:   NOP   0;
      A     #P.KB2_Istnieje;
      AN    #P.KB2_Wpis;
      JCN   z1;
      L     #id_Wartosc_KB2;
      T     #Help_Dint;
      AN    #P.KB2_Wpis;
      =     #Temp_Wpis_KB2;
      JU    x0;
z1:   NOP   0;
      A     #P.I1_Istnieje;
      AN    #P.I1_Wpis;
      JCN   z2;
      L     #id_Wartosc_I1;
      T     #Help_Dint;
      AN    #P.I1_Wpis;
      =     #Temp_Wpis_I1;
      JU    x0;
z2:   NOP   0;
      A     #P.I2_Istnieje;
      AN    #P.I2_Wpis;
      JCN   z3;
      L     #id_Wartosc_I2;
      T     #Help_Dint;
      AN    #P.I2_Wpis;
      =     #Temp_Wpis_I2;
      JU    x0;
z3:   NOP   0;
      A     #P.I3_Istnieje;
      AN    #P.I3_Wpis;
      JCN   z4;
      L     #id_Wartosc_I3;
      T     #Help_Dint;
      AN    #P.I3_Wpis;
      =     #Temp_Wpis_I3;
      JU    x0;
z4:   NOP   0;
//wartosc wagowa
//***sprawdzenie pozycji 0**********************
x0:   L     LW 10;
      L     #Wpis._0_dbw2_War_Wagowa;
      >I;
      A(;
      O     #Temp_Wpis_KB1;
      O     #Temp_Wpis_KB2;
      O     #Temp_Wpis_I1;
      O     #Temp_Wpis_I2;
      O     #Temp_Wpis_I3;
      );
      JCN   k0;
//zrobienie miejsca na nowy rekord
//***pozycja 4-5
      L     LD 28;
      T     LD 32;
//***pozycja 3-4
      L     LD 24;
      T     LD 28;
//***pozycja 2-3
      L     LD 20;
      T     LD 24;
//***pozycja 1-2
      L     LD 16;
      T     LD 20;
//***pozycja 0-1
      L     LD 12;
      T     LD 16;
      L     #Help_Dint;	//id_wartosc
      T     LD 12;	//element
//Potwierdzenie wpisania
      A     #Temp_Wpis_KB1;
      S     #P.KB1_Wpis;
      A     #Temp_Wpis_KB2;
      S     #P.KB2_Wpis;
      A     #Temp_Wpis_I1;
      S     #P.I1_Wpis;
      A     #Temp_Wpis_I2;
      S     #P.I2_Wpis;
      A     #Temp_Wpis_I3;
      S     #P.I3_Wpis;
      SET;
      R     #Temp_Wpis_KB1;
      R     #Temp_Wpis_KB2;
      R     #Temp_Wpis_I1;
      R     #Temp_Wpis_I2;
      R     #Temp_Wpis_I3;
k0:   NOP   0;
//***sprawdzenie pozycji 1**********************
      L     LW 10;
      L     #Wpis._1_dbw6_War_Wagowa;
      >I;
      A(;
      O     #Temp_Wpis_KB1;
      O     #Temp_Wpis_KB2;
      O     #Temp_Wpis_I1;
      O     #Temp_Wpis_I2;
      O     #Temp_Wpis_I3;
      );
      JCN   k1;
//***pozycja 4-5
      L     LD 28;
      T     LD 32;
//***pozycja 3-4
      L     LD 24;
      T     LD 28;
//***pozycja 2-3
      L     LD 20;
      T     LD 24;
//***pozycja 1-2
      L     LD 16;
      T     LD 20;
      L     #Help_Dint;	//id_wartosc
      T     LD 16;	//element
//Potwierdzenie wpisania
      A     #Temp_Wpis_KB1;
      S     #P.KB1_Wpis;
      A     #Temp_Wpis_KB2;
      S     #P.KB2_Wpis;
      A     #Temp_Wpis_I1;
      S     #P.I1_Wpis;
      A     #Temp_Wpis_I2;
      S     #P.I2_Wpis;
      A     #Temp_Wpis_I3;
      S     #P.I3_Wpis;
      SET;
      R     #Temp_Wpis_KB1;
      R     #Temp_Wpis_KB2;
      R     #Temp_Wpis_I1;
      R     #Temp_Wpis_I2;
      R     #Temp_Wpis_I3;
k1:   NOP   0;
//***sprawdzenie pozycji 2
      L     LW 10;
      L     #Wpis._2_dbw10_War_Wagowa;
      >I;
      A(;
      O     #Temp_Wpis_KB1;
      O     #Temp_Wpis_KB2;
      O     #Temp_Wpis_I1;
      O     #Temp_Wpis_I2;
      O     #Temp_Wpis_I3;
      );
      JCN   k2;
//***pozycja 4-5
      L     LD 28;
      T     LD 32;
//***pozycja 3-4
      L     LD 24;
      T     LD 28;
//***pozycja 2-3
      L     LD 20;
      T     LD 24;
      L     #Help_Dint;	//id_wartosc
      T     LD 20;	//element
//Potwierdzenie wpisania
      A     #Temp_Wpis_KB1;
      S     #P.KB1_Wpis;
      A     #Temp_Wpis_KB2;
      S     #P.KB2_Wpis;
      A     #Temp_Wpis_I1;
      S     #P.I1_Wpis;
      A     #Temp_Wpis_I2;
      S     #P.I2_Wpis;
      A     #Temp_Wpis_I3;
      S     #P.I3_Wpis;
      SET;
      R     #Temp_Wpis_KB1;
      R     #Temp_Wpis_KB2;
      R     #Temp_Wpis_I1;
      R     #Temp_Wpis_I2;
      R     #Temp_Wpis_I3;
k2:   NOP   0;
//***sprawdzenie pozycji 3
      L     LW 10;
      L     #Wpis._3_dbw14_War_Wagowa;
      >I;
      A(;
      O     #Temp_Wpis_KB1;
      O     #Temp_Wpis_KB2;
      O     #Temp_Wpis_I1;
      O     #Temp_Wpis_I2;
      O     #Temp_Wpis_I3;
      );
      JCN   k3;
//***pozycja 4-5
      L     LD 28;
      T     LD 32;
//***pozycja 3-4
      L     LD 24;
      T     LD 28;
      L     #Help_Dint;	//id_wartosc
      T     LD 24;	//element
//Potwierdzenie wpisania
      A     #Temp_Wpis_KB1;
      S     #P.KB1_Wpis;
      A     #Temp_Wpis_KB2;
      S     #P.KB2_Wpis;
      A     #Temp_Wpis_I1;
      S     #P.I1_Wpis;
      A     #Temp_Wpis_I2;
      S     #P.I2_Wpis;
      A     #Temp_Wpis_I3;
      S     #P.I3_Wpis;
      SET;
      R     #Temp_Wpis_KB1;
      R     #Temp_Wpis_KB2;
      R     #Temp_Wpis_I1;
      R     #Temp_Wpis_I2;
      R     #Temp_Wpis_I3;
k3:   NOP   0;
//***sprawdzenie pozycji 4
      L     LW 10;
      L     #Wpis._4_dbw18_War_Wagowa;
      >I;
      A(;
      O     #Temp_Wpis_KB1;
      O     #Temp_Wpis_KB2;
      O     #Temp_Wpis_I1;
      O     #Temp_Wpis_I2;
      O     #Temp_Wpis_I3;
      );
      JCN   k4;
//***pozycja 4-5
      L     LD 28;
      T     LD 32;
      L     #Help_Dint;	//id_wartosc
      T     LD 28;	//element
//Potwierdzenie wpisania
      A     #Temp_Wpis_KB1;
      S     #P.KB1_Wpis;
      A     #Temp_Wpis_KB2;
      S     #P.KB2_Wpis;
      A     #Temp_Wpis_I1;
      S     #P.I1_Wpis;
      A     #Temp_Wpis_I2;
      S     #P.I2_Wpis;
      A     #Temp_Wpis_I3;
      S     #P.I3_Wpis;
      SET;
      R     #Temp_Wpis_KB1;
      R     #Temp_Wpis_KB2;
      R     #Temp_Wpis_I1;
      R     #Temp_Wpis_I2;
      R     #Temp_Wpis_I3;
k4:   NOP   0;
//***sprawdzenie pozycji 5
      L     LW 10;
      L     #Wpis._5_dbw22_War_Wagowa;
      >I;
      A(;
      O     #Temp_Wpis_KB1;
      O     #Temp_Wpis_KB2;
      O     #Temp_Wpis_I1;
      O     #Temp_Wpis_I2;
      O     #Temp_Wpis_I3;
      );
      JCN   k5;
//***pozycja 4-5
      L     #Help_Dint;	//id_wartosc
      T     LD 32;	//element
//Potwierdzenie wpisania
      A     #Temp_Wpis_KB1;
      S     #P.KB1_Wpis;
      A     #Temp_Wpis_KB2;
      S     #P.KB2_Wpis;
      A     #Temp_Wpis_I1;
      S     #P.I1_Wpis;
      A     #Temp_Wpis_I2;
      S     #P.I2_Wpis;
      A     #Temp_Wpis_I3;
      S     #P.I3_Wpis;
      SET;
      R     #Temp_Wpis_KB1;
      R     #Temp_Wpis_KB2;
      R     #Temp_Wpis_I1;
      R     #Temp_Wpis_I2;
      R     #Temp_Wpis_I3;
k5:   NOP   0;
NETWORK
TITLE =
NETWORK
TITLE =
//Sprawdzenie czy wpisy nie sa zerami
      L     #Wpis._0_dbw2_War_Wagowa;
      L     0;
      >I;
      =     #P.Wpis_0_istnieje;
//1
      L     #Wpis._1_dbw6_War_Wagowa;
      L     0;
      >I;
      =     #P.Wpis_1_istnieje;
//2
      L     #Wpis._2_dbw10_War_Wagowa;
      L     0;
      >I;
      =     #P.Wpis_2_istnieje;
//3
      L     #Wpis._3_dbw14_War_Wagowa;
      L     0;
      >I;
      =     #P.Wpis_3_istnieje;
//4
      L     #Wpis._4_dbw18_War_Wagowa;
      L     0;
      >I;
      =     #P.Wpis_4_istnieje;
//5
      L     #Wpis._5_dbw22_War_Wagowa;
      L     0;
      >I;
      =     #P.Wpis_5_istnieje;
NETWORK
TITLE =
//Przesowanie rejestrow w gore i dol
//toggle 0 i 1 
      A(;
      O     #i_Poz_5_Down;
      O     #i_Poz_4_Up;
      );
      FP    #P.edge_1;
      A     #P.Wpis_0_istnieje;
      A     #P.Wpis_1_istnieje;
      JCN   w0;
      L     LW 12;
      T     #Help_Int_2;
      L     #Wpis._0_dbw2_War_Wagowa;
      T     LW 12;
      L     #Help_Int_2;
      T     #Wpis._0_dbw2_War_Wagowa;
w0:   NOP   0;
//toggle 1 i 2  
      A(;
      O     #i_Poz_4_Down;
      O     #i_Poz_3_Up;
      );
      FP    #P.edge_2;
      A     #P.Wpis_1_istnieje;
      A     #P.Wpis_2_istnieje;
      JCN   w1;
      L     #Wpis._0_dbw2_War_Wagowa;
      T     #Help_Int_2;
      L     #Wpis._1_dbw6_War_Wagowa;
      T     #Wpis._0_dbw2_War_Wagowa;
      L     #Help_Int_2;
      T     #Wpis._1_dbw6_War_Wagowa;
w1:   NOP   0;
//toggle 2 i 3  
      A(;
      O     #i_Poz_3_Down;
      O     #i_Poz_2_Up;
      );
      FP    #P.edge_3;
      A     #P.Wpis_2_istnieje;
      A     #P.Wpis_3_istnieje;
      JCN   w2;
      L     #Wpis._1_dbw6_War_Wagowa;
      T     #Help_Int_2;
      L     #Wpis._2_dbw10_War_Wagowa;
      T     #Wpis._1_dbw6_War_Wagowa;
      L     #Help_Int_2;
      T     #Wpis._2_dbw10_War_Wagowa;
w2:   NOP   0;
//toggle 3 i 4  
      A(;
      O     #i_Poz_2_Down;
      O     #i_Poz_1_Up;
      );
      FP    #P.edge_4;
      A     #P.Wpis_3_istnieje;
      A     #P.Wpis_4_istnieje;
      JCN   w3;
      L     #Wpis._2_dbw10_War_Wagowa;
      T     #Help_Int_2;
      L     #Wpis._3_dbw14_War_Wagowa;
      T     #Wpis._2_dbw10_War_Wagowa;
      L     #Help_Int_2;
      T     #Wpis._3_dbw14_War_Wagowa;
w3:   NOP   0;
NETWORK
TITLE =
      L     #P;
      T     #iow_Help_DWord;
//Zaladowanie pakietu danych
      CALL  "BLKMOV" (
           SRCBLK                   := #Wpis,
           RET_VAL                  := #Help_Blok_Move,
           DSTBLK                   := "Key_DB".Wpis);
END_FUNCTION

FUNCTION "Wozek_Jezdny_Kolejka" : VOID	// FC 600
//Nalezy w HMI dopisac brakujace kody obslugi jazdy (kod 17 i kod 18)
//
VERSION : 0.1
BEGIN
NETWORK
TITLE =
//Ten Network celowo jest wolny
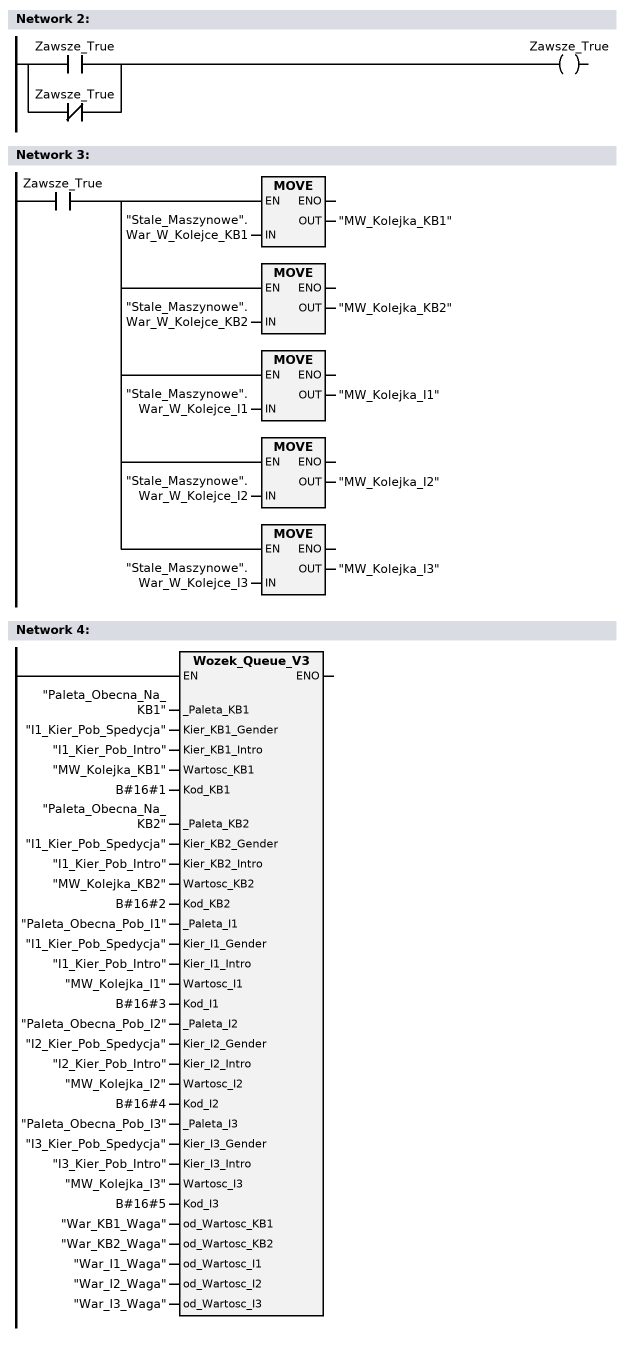
NETWORK
TITLE =
      O     "Zawsze_True";
      ON    "Zawsze_True";
      =     "Zawsze_True";
NETWORK
TITLE =
//Wartosc danej pozycji w kolejce
      A     "Zawsze_True";
      =     L 0.0;
      A     L 0.0;
      JNB   _001;
      L     "Stale_Maszynowe".War_W_Kolejce_KB1;
      T     "MW_Kolejka_KB1";
_001: NOP   0;
      A     L 0.0;
      JNB   _002;
      L     "Stale_Maszynowe".War_W_Kolejce_KB2;
      T     "MW_Kolejka_KB2";
_002: NOP   0;
      A     L 0.0;
      JNB   _003;
      L     "Stale_Maszynowe".War_W_Kolejce_I1;
      T     "MW_Kolejka_I1";
_003: NOP   0;
      A     L 0.0;
      JNB   _004;
      L     "Stale_Maszynowe".War_W_Kolejce_I2;
      T     "MW_Kolejka_I2";
_004: NOP   0;
      A     L 0.0;
      JNB   _005;
      L     "Stale_Maszynowe".War_W_Kolejce_I3;
      T     "MW_Kolejka_I3";
_005: NOP   0;
NETWORK
TITLE =
//Dostep do kolejki jazdy wozkiem
//MB620-kierunek intro(0),spedycja(1)
//MB621-Kod mszyny np KB1-1
//MW622-Wartosc wagowa (Pobrana ze stalych maszynowych)
//
//
//
      CALL  "Wozek_Queue_V3" (
           _Paleta_KB1              := "Paleta_Obecna_Na_KB1",
           Kier_KB1_Gender          := "I1_Kier_Pob_Spedycja",
           Kier_KB1_Intro           := "I1_Kier_Pob_Intro",
           Wartosc_KB1              := "MW_Kolejka_KB1",
           Kod_KB1                  := B#16#1,
           _Paleta_KB2              := "Paleta_Obecna_Na_KB2",
           Kier_KB2_Gender          := "I1_Kier_Pob_Spedycja",
           Kier_KB2_Intro           := "I1_Kier_Pob_Intro",
           Wartosc_KB2              := "MW_Kolejka_KB2",
           Kod_KB2                  := B#16#2,
           _Paleta_I1               := "Paleta_Obecna_Pob_I1",
           Kier_I1_Gender           := "I1_Kier_Pob_Spedycja",
           Kier_I1_Intro            := "I1_Kier_Pob_Intro",
           Wartosc_I1               := "MW_Kolejka_I1",
           Kod_I1                   := B#16#3,
           _Paleta_I2               := "Paleta_Obecna_Pob_I2",
           Kier_I2_Gender           := "I2_Kier_Pob_Spedycja",
           Kier_I2_Intro            := "I2_Kier_Pob_Intro",
           Wartosc_I2               := "MW_Kolejka_I2",
           Kod_I2                   := B#16#4,
           _Paleta_I3               := "Paleta_Obecna_Pob_I3",
           Kier_I3_Gender           := "I3_Kier_Pob_Spedycja",
           Kier_I3_Intro            := "I3_Kier_Pob_Intro",
           Wartosc_I3               := "MW_Kolejka_I3",
           Kod_I3                   := B#16#5,
           od_Wartosc_KB1           := "War_KB1_Waga",
           od_Wartosc_KB2           := "War_KB2_Waga",
           od_Wartosc_I1            := "War_I1_Waga",
           od_Wartosc_I2            := "War_I2_Waga",
           od_Wartosc_I3            := "War_I3_Waga");
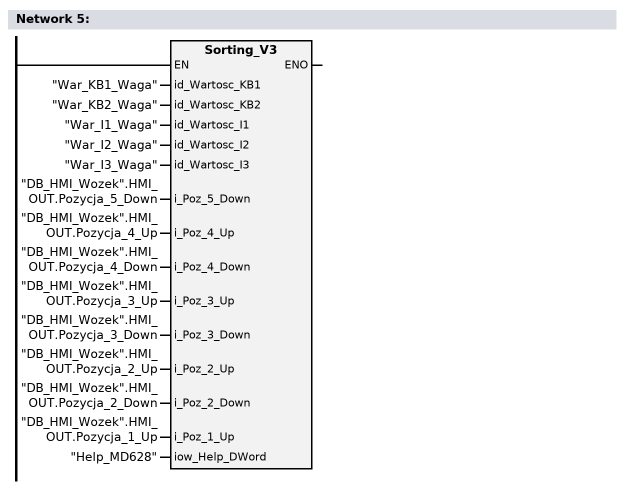
NETWORK
TITLE =
//Zbudowanie rekordu
      CALL  "Sorting_V3" (
           id_Wartosc_KB1           := "War_KB1_Waga",
           id_Wartosc_KB2           := "War_KB2_Waga",
           id_Wartosc_I1            := "War_I1_Waga",
           id_Wartosc_I2            := "War_I2_Waga",
           id_Wartosc_I3            := "War_I3_Waga",
           i_Poz_5_Down             := "DB_HMI_Wozek".HMI_OUT.Pozycja_5_Down,
           i_Poz_4_Up               := "DB_HMI_Wozek".HMI_OUT.Pozycja_4_Up,
           i_Poz_4_Down             := "DB_HMI_Wozek".HMI_OUT.Pozycja_4_Down,
           i_Poz_3_Up               := "DB_HMI_Wozek".HMI_OUT.Pozycja_3_Up,
           i_Poz_3_Down             := "DB_HMI_Wozek".HMI_OUT.Pozycja_3_Down,
           i_Poz_2_Up               := "DB_HMI_Wozek".HMI_OUT.Pozycja_2_Up,
           i_Poz_2_Down             := "DB_HMI_Wozek".HMI_OUT.Pozycja_2_Down,
           i_Poz_1_Up               := "DB_HMI_Wozek".HMI_OUT.Pozycja_1_Up,
           iow_Help_DWord           := "Help_MD628");
END_FUNCTION

FUNCTION "Send_Data" : VOID	// FC 700
//Funkcja Send_Data odpowiada za zapis duzej ilosci danych  z drugiego waskim 
//kanalem informacyjnym (kilku bajtowym). Funkcja 
//skonstruowana glownie do przesylu parametrow.
//
//Read_Data pracuje w parze z Share_Data
//
//Poszczegolne kroki w wysylaniu i odbieraniu
//
//i_Rozpocznij_Transmisje
//o_zadanie_transmisji     --> i_transmisja_ustanowiona
//ow_Nr_Bloku_Pobieranego  --> i_Blok_Pobierany_Zerezerwowany
//o_zadanie_danych         --> i_przesylanie_danych
//                         --> i_koniec_przesylania
//
//
//
//Po kazdej przeslanej danej musi dosjsc do inwersji bitu toggle
VERSION : 0.1
VAR_INPUT
  i_Reset : BOOL ;	//Reset Transmisji
  i_Rozpocznij_Transmisje : BOOL ;	//Wyslij dane (Wejscie aktywne na zbocze)
  i_Transmisja_Ustanowiona : BOOL ;	//Odpowiedz na zadanie transmisji
  i_Blok_Zew_Zarezerwowany : BOOL ;	//Potwierdzenie rezerwacji bloku w drugim urzadzeniu
  i_Przesylanie_Danych : BOOL ;	//Przesylanie w toku
  iw_Nr_Bloku_Nadpisu : INT ;	//Nr przesylanego bloku danych
  iw_Nr_Bloku_Poboru : INT ;	//Nr bloku gdzie dane sa zapisane
  iw_Ilosc_Max_Rekordow : INT ;	//Ilosc pobieranych rekordow
  iw_Rekord_Powracajacy : INT ;	//Potwierdzenie nr rekordu
END_VAR
VAR_OUTPUT
  o_Zadanie_Transmisji : BOOL ;	//Ustanowienie transmisji
  o_Zadanie_Danych : BOOL ;	//Zadanie wyslania indeksu danych
  o_Koniec_Nadawania : BOOL ;	//Sygnal opadajacy
  ow_Nr_Bloku_Nadpisu : INT ;
  ow_Nr_Rekordu : INT ;
  ow_Kanal_Nadawania : INT ;	//Kanal wysylania
END_VAR
VAR_IN_OUT
  io_Help_Word : WORD ;
  iow_NR_Petli : INT ;	//Nr petli danych
END_VAR
VAR_TEMP
  Przesylanie_Aktywne : BOOL ;
  L_Rozpocznij_Transfer : BOOL ;
  Zbocze_1 : BOOL ;
  Temp_Byte : BYTE ;
  Help_Word_2 : WORD ;
  L_NR_Bloku_Zapisu : WORD ;
  L_Nr_Recordu : DWORD ;
  L_DW_Licznik_Rekordow : DWORD ;
END_VAR
BEGIN
NETWORK
TITLE =
//Ten Network celowo jest wolny
NETWORK
TITLE =
//Pobranie zmiennych pomocniczych
      L     #io_Help_Word;
      T     #Help_Word_2;
NETWORK
TITLE =
//Pobierz nazwe bloku kopiowanego
      L     #iw_Nr_Bloku_Poboru;	// Nr bloku db
      T     #L_NR_Bloku_Zapisu;
      OPN   DB [#L_NR_Bloku_Zapisu];	// Otwarcie db
NETWORK
TITLE =
//Rzadanie transmisji
//
      A     #i_Rozpocznij_Transmisje;
      FP    #Zbocze_1;
      S     #L_Rozpocznij_Transfer;
      S     #o_Koniec_Nadawania;
      JCN   zer;
      L     0;
      T     #iow_NR_Petli;
zer:  NOP   0;
      A     #L_Rozpocznij_Transfer;
      =     #o_Zadanie_Transmisji;
NETWORK
TITLE =
//Przeslanie nazwy bloku 
//Przeslanie nazwy bloku odbierania danych. Potwierdzeni wraca bitem
//blok_Odb_Zarezerwowany
      A     #L_Rozpocznij_Transfer;
      A     #i_Transmisja_Ustanowiona;
      JCN   et_1;
      L     #iw_Nr_Bloku_Nadpisu;
      T     #ow_Nr_Bloku_Nadpisu;
      JU    et_2;
et_1: NOP   0;
      L     0;
      T     #ow_Nr_Bloku_Nadpisu;
et_2: NOP   0;
NETWORK
TITLE =
//Przeslanie Pierwszego podwojenego slowa w celu nawiazania komunikacji
      A     #L_Rozpocznij_Transfer;
      A     #i_Blok_Zew_Zarezerwowany;
      A     #i_Transmisja_Ustanowiona;
      =     #o_Zadanie_Danych;
NETWORK
TITLE =
//Otrzymanie potwierdzenia
      A     #L_Rozpocznij_Transfer;
      A     #i_Blok_Zew_Zarezerwowany;
      A     #i_Transmisja_Ustanowiona;
      A     #i_Przesylanie_Danych;
      =     #Przesylanie_Aktywne;
//Wylicz nr rekordu
      L     #iow_NR_Petli;
      L     2;
      *I;
      ITD;
      SLD   3;
      T     #L_DW_Licznik_Rekordow;
      L     #iow_NR_Petli;
      T     #ow_Nr_Rekordu;
// podlicz rekordy
      A(;
      L     #iow_NR_Petli;
      L     #iw_Rekord_Powracajacy;
      ==I;
      );
      A     #Przesylanie_Aktywne;
      JCN   et_3;
      L     DBW [#L_DW_Licznik_Rekordow];	//h
      T     #ow_Kanal_Nadawania;
      L     #iow_NR_Petli;
      L     1;
      +I;
      T     #iow_NR_Petli;
et_3: NOP   0;
//Zakoncz gdy koniec iteracji
      O(;
      L     #iow_NR_Petli;
      L     #iw_Ilosc_Max_Rekordow;
      >=I;
      );
      O     #i_Reset;
      JCN   d0;
      L     0;
      T     #iw_Ilosc_Max_Rekordow;
      SET;
      R     #L_Rozpocznij_Transfer;
      R     #o_Koniec_Nadawania;
d0:   NOP   0;
NETWORK
TITLE =
//Zapis bitow przejsciowych
      L     #Help_Word_2;
      T     #io_Help_Word;
END_FUNCTION

FUNCTION "Receive_Data" : VOID	// FC 701
//Funkcja Share_Data udostepnia dane funkcji Read_Data. Sluzy do odczytu 
//parametrow z oddalonego urzadzenia przez waski kilku-bajtowy kanal 
//komunikacyjny.
//Poszczegolne kroki w wysylaniu i odbieraniu
//
//i_zadanie_transmisji     --> o_transmisja_ustanowiona
//iw_Nr_Bloku_Pobieranego  --> o_Blok_Pobierany_Zarezerwowany
//i_zadanie_danych         --> o_przesylanie_danych
//                         --> o_koniec_przesylania
//
//Po kazdej przeslanej danej musi dosjsc do inwersji bitu toggle
VERSION : 0.1
VAR_INPUT
  i_Zadanie_Transmisji : BOOL ;	//Ustanowienie transmisji
  i_Zadanie_Danych : BOOL ;	//Zadanie wyslania indeksu danych
  iw_Nr_Bloku_Nadpisu : INT ;
  iw_Nr_Rekordu : INT ;
  iw_Kanal_Odbioru : INT ;
END_VAR
VAR_OUTPUT
  o_Transmisja_Ustanowiona : BOOL ;	//Odpowiedz na zadanie transmisji
  o_Blok_Odb_Zarezerwowany : BOOL ;	//Potwierdzenie rezerwacji bloku
  o_Przesylanie_Danych : BOOL ;	//Przesylanie w toku
  ow_Rekord_Powracajacy : INT ;
END_VAR
VAR_IN_OUT
  io_Help_Word : WORD ;
END_VAR
VAR_TEMP
  Temp_Bool_1 : BOOL ;
  Temp_Byte : BYTE ;
  Help_Word_2 : WORD ;
  L_NR_Bloku_Danych : WORD ;
  L_Liczba_Rekordow : INT ;
  L_DW_Licznik_Rekordow : DWORD ;
END_VAR
BEGIN
NETWORK
TITLE =
//Ten Network celowo jest wolny
NETWORK
TITLE =
//Pobranie zmiennych pomocniczych
      L     #io_Help_Word;
      T     #Help_Word_2;
NETWORK
TITLE =
//Rzadanie transmisji
//
      A     #i_Zadanie_Transmisji;
      =     #o_Transmisja_Ustanowiona;
NETWORK
TITLE =
//Reset licznika rekordow
      A     #i_Zadanie_Transmisji;
      AN    #i_Zadanie_Danych;
      JCN   et_1;
      L     0;
      T     #ow_Rekord_Powracajacy;
et_1: NOP   0;
NETWORK
TITLE =
//Pobierz nazwe bloku kopiowanego
// sprawdzenie czy blok rozny od 0
      L     #iw_Nr_Bloku_Nadpisu;
      T     #L_NR_Bloku_Danych;
      L     0;
      <>I;
      =     #o_Blok_Odb_Zarezerwowany;
      A     #i_Zadanie_Transmisji;
      A     #i_Zadanie_Danych;
      =     #o_Przesylanie_Danych;
      AN    #o_Blok_Odb_Zarezerwowany;
      JC    end;
//Blok pobierany
      OPN   DB [#L_NR_Bloku_Danych];	// Otwarcie db
NETWORK
TITLE =
//Przeslanie Pierwszego podwojenego slowa w celu nawiazania komunikacji
// zamiania na double 
      L     #iw_Nr_Rekordu;
      L     2;
      *I;
      ITD;
      SLD   3;
      T     #L_DW_Licznik_Rekordow;
//Transmisja
      A     #o_Przesylanie_Danych;
      JCN   et_4;
      L     #iw_Kanal_Odbioru;
      T     DBW [#L_DW_Licznik_Rekordow];
      L     #iw_Nr_Rekordu;
      T     #ow_Rekord_Powracajacy;
et_4: NOP   0;
end:  NOP   0;
NETWORK
TITLE =
//Zapis bitow przejsciowych
      L     #Help_Word_2;
      T     #io_Help_Word;
      BEU;
END_FUNCTION

FUNCTION "Read_Data" : VOID	// FC 702
//Funkcja Read_Data odpowiada za odczyt duzej ilosci danych  z drugiego waskim 
//kanalem informacyjnym (kilku bajtowym). Funkcja 
//skonstruowana glownie do przesylu parametrow.
//
//Read_Data pracuje w parze z Share_Data
//
//Poszczegolne kroki w wysylaniu i odbieraniu
//
//i_Rozpocznij_Transmisje
//o_zadanie_transmisji     --> i_transmisja_ustanowiona
//ow_Nr_Bloku_Pobieranego  --> i_Blok_Pobierany_Zerezerwowany
//o_zadanie_danych         --> i_przesylanie_danych
//                         --> i_koniec_przesylania
//
//
//
//Po kazdej przeslanej danej musi dosjsc do inwersji bitu toggle
VERSION : 0.1
VAR_INPUT
  i_Reset : BOOL ;	//Reset Transmisji
  i_Rozpocznij_Transmisje : BOOL ;	//Wyslij dane (Wejscie aktywne na zbocze)
  i_Transmisja_Ustanowiona : BOOL ;	//Odpowiedz na zadanie transmisji
  i_Blok_Zew_Zarezerwowany : BOOL ;	//Potwierdzenie rezerwacji bloku w drugim urzadzeniu
  i_Przesylanie_Danych : BOOL ;	//Przesylanie w toku
  iw_Nr_Bloku_Pobieranego : INT ;	//Nr przesylanego bloku danych
  iw_Nr_Bloku_Zapisu : INT ;	//Nr bloku gdzie dane sa zapisane
  iw_Kanal_Odbierania : INT ;	//Kanal danych pobieranych
  iw_Ilosc_Max_Rekordow : INT ;	//Ilosc pobieranych rekordow
  iw_Rekord_Powracajacy : INT ;	//Potwierdzenie nr rekordu
END_VAR
VAR_OUTPUT
  o_Zadanie_Transmisji : BOOL ;	//Ustanowienie transmisji
  o_Zadanie_Danych : BOOL ;	//Zadanie wyslania indeksu danych
  o_Koniec_Nadawania : BOOL ;	//Sygnal opadajacy
  ow_Nr_Bloku_Pobieranego : INT ;
  ow_Nr_Rekordu : INT ;
END_VAR
VAR_IN_OUT
  io_Help_Word : WORD ;
  iow_NR_Petli : INT ;	//Nr petli danych
END_VAR
VAR_TEMP
  Przesylanie_Aktywne : BOOL ;
  L_Rozpocznij_Transfer : BOOL ;
  Zbocze_1 : BOOL ;
  Temp_Byte : BYTE ;
  Help_Word_2 : WORD ;
  L_NR_Bloku_Zapisu : WORD ;
  L_Nr_Recordu : DWORD ;
  L_DW_Licznik_Rekordow : DWORD ;
END_VAR
BEGIN
NETWORK
TITLE =
//Ten Network celowo jest wolny
NETWORK
TITLE =
//Pobranie zmiennych pomocniczych
      L     #io_Help_Word;
      T     #Help_Word_2;
NETWORK
TITLE =
//Pobierz nazwe bloku kopiowanego
      L     #iw_Nr_Bloku_Zapisu;	// Nr bloku db
      T     #L_NR_Bloku_Zapisu;
      OPN   DB [#L_NR_Bloku_Zapisu];	// Otwarcie db
NETWORK
TITLE =
//Rzadanie transmisji
//
      A     #i_Rozpocznij_Transmisje;
      FP    #Zbocze_1;
      S     #L_Rozpocznij_Transfer;
      S     #o_Koniec_Nadawania;
      JCN   zer;
      L     0;
      T     #iow_NR_Petli;
zer:  NOP   0;
      A     #L_Rozpocznij_Transfer;
      =     #o_Zadanie_Transmisji;
NETWORK
TITLE =
//Przeslanie nazwy bloku 
//Przeslanie nazwy bloku odbierania danych. Potwierdzeni wraca bitem
//blok_Odb_Zarezerwowany
      A     #L_Rozpocznij_Transfer;
      A     #i_Transmisja_Ustanowiona;
      JCN   et_1;
      L     #iw_Nr_Bloku_Pobieranego;
      T     #ow_Nr_Bloku_Pobieranego;
      JU    et_2;
et_1: NOP   0;
      L     0;
      T     #ow_Nr_Bloku_Pobieranego;
et_2: NOP   0;
NETWORK
TITLE =
//Przeslanie Pierwszego podwojenego slowa w celu nawiazania komunikacji
      A     #L_Rozpocznij_Transfer;
      A     #i_Blok_Zew_Zarezerwowany;
      A     #i_Transmisja_Ustanowiona;
      =     #o_Zadanie_Danych;
NETWORK
TITLE =
//Otrzymanie potwierdzenia
      A     #L_Rozpocznij_Transfer;
      A     #i_Blok_Zew_Zarezerwowany;
      A     #i_Transmisja_Ustanowiona;
      A     #i_Przesylanie_Danych;
      =     #Przesylanie_Aktywne;
//Wylicz nr rekordu
      L     #iow_NR_Petli;
      L     2;
      *I;
      ITD;
      SLD   3;
      T     #L_DW_Licznik_Rekordow;
      L     #iow_NR_Petli;
      T     #ow_Nr_Rekordu;
// podlicz rekordy
      A(;
      L     #iow_NR_Petli;
      L     #iw_Rekord_Powracajacy;
      ==I;
      );
      A     #Przesylanie_Aktywne;
      JCN   et_3;
      L     #iw_Kanal_Odbierania;
      T     DBW [#L_DW_Licznik_Rekordow];	//Zapisanie danych
      L     #iow_NR_Petli;
      L     1;
      +I;
      T     #iow_NR_Petli;
et_3: NOP   0;
//Zakoncz gdy koniec iteracji
      O(;
      L     #iow_NR_Petli;
      L     #iw_Ilosc_Max_Rekordow;
      >=I;
      );
      O     #i_Reset;
      JCN   d0;
      L     0;
      T     #iw_Ilosc_Max_Rekordow;
      SET;
      R     #L_Rozpocznij_Transfer;
      R     #o_Koniec_Nadawania;
d0:   NOP   0;
NETWORK
TITLE =
//Zapis bitow przejsciowych
      L     #Help_Word_2;
      T     #io_Help_Word;
END_FUNCTION

FUNCTION "Share_Data" : VOID	// FC 703
//Funkcja Share_Data udostepnia dane funkcji Read_Data. Sluzy do odczytu 
//parametrow z oddalonego urzadzenia przez waski kilku-bajtowy kanal 
//komunikacyjny.
//Poszczegolne kroki w wysylaniu i odbieraniu
//
//i_zadanie_transmisji     --> o_transmisja_ustanowiona
//iw_Nr_Bloku_Pobieranego  --> o_Blok_Pobierany_Zarezerwowany
//i_zadanie_danych         --> o_przesylanie_danych
//                         --> o_koniec_przesylania
//
//Po kazdej przeslanej danej musi dosjsc do inwersji bitu toggle
VERSION : 0.1
VAR_INPUT
  i_Zadanie_Transmisji : BOOL ;	//Ustanowienie transmisji
  i_Zadanie_Danych : BOOL ;	//Zadanie wyslania indeksu danych
  iw_Nr_Bloku_Pobieranego : INT ;
  iw_Nr_Rekordu : INT ;
END_VAR
VAR_OUTPUT
  o_Transmisja_Ustanowiona : BOOL ;	//Odpowiedz na zadanie transmisji
  o_Blok_Odb_Zarezerwowany : BOOL ;	//Potwierdzenie rezerwacji bloku
  o_Przesylanie_Danych : BOOL ;	//Przesylanie w toku
  ow_Kanal_Pobierania : INT ;	//Dane ktore sa udostepniane
  ow_Rekord_Powracajacy : INT ;
END_VAR
VAR_IN_OUT
  io_Help_Word : WORD ;
END_VAR
VAR_TEMP
  Temp_Bool_1 : BOOL ;
  Temp_Byte : BYTE ;
  Help_Word_2 : WORD ;
  L_NR_Bloku_Danych : WORD ;
  L_Liczba_Rekordow : INT ;
  L_DW_Licznik_Rekordow : DWORD ;
END_VAR
BEGIN
NETWORK
TITLE =
//Ten Network celowo jest wolny
NETWORK
TITLE =
//Pobranie zmiennych pomocniczych
      L     #io_Help_Word;
      T     #Help_Word_2;
NETWORK
TITLE =
//Rzadanie transmisji
//
      A     #i_Zadanie_Transmisji;
      =     #o_Transmisja_Ustanowiona;
NETWORK
TITLE =
//Reset licznika rekordow
      A     #i_Zadanie_Transmisji;
      AN    #i_Zadanie_Danych;
      JCN   et_1;
      L     0;
      T     #ow_Rekord_Powracajacy;
et_1: NOP   0;
NETWORK
TITLE =
//Pobierz nazwe bloku kopiowanego
// sprawdzenie czy blok rozny od 0
      L     #iw_Nr_Bloku_Pobieranego;
      T     #L_NR_Bloku_Danych;
      L     0;
      <>I;
      =     #o_Blok_Odb_Zarezerwowany;
      A     #i_Zadanie_Transmisji;
      A     #i_Zadanie_Danych;
      =     #o_Przesylanie_Danych;
      AN    #o_Blok_Odb_Zarezerwowany;
      JC    end;
//Blok pobierany
      OPN   DB [#L_NR_Bloku_Danych];	// Otwarcie db
NETWORK
TITLE =
//Przeslanie Pierwszego podwojenego slowa w celu nawiazania komunikacji
// zamiania na double 
      L     #iw_Nr_Rekordu;
      L     2;
      *I;
      ITD;
      SLD   3;
      T     #L_DW_Licznik_Rekordow;
//Transmisja
      A     #o_Przesylanie_Danych;
      JCN   et_4;
      L     DBW [#L_DW_Licznik_Rekordow];
      T     #ow_Kanal_Pobierania;
      L     #iw_Nr_Rekordu;
      T     #ow_Rekord_Powracajacy;
et_4: NOP   0;
end:  NOP   0;
NETWORK
TITLE =
//Zapis bitow przejsciowych
      L     #Help_Word_2;
      T     #io_Help_Word;
      BEU;
END_FUNCTION

DATA_BLOCK DB 100
VERSION : 0.1
  STRUCT
   DB_VAR : INT ;	//Temporary placeholder variable
   DB_VAR1 : INT ;	//Temporary placeholder variable
   DB_VAR2 : INT ;	//Temporary placeholder variable
   DB_VAR3 : INT ;	//Temporary placeholder variable
   DB_VAR4 : INT ;	//Temporary placeholder variable
   DB_VAR5 : INT ;	//Temporary placeholder variable
   DB_VAR6 : INT ;	//Temporary placeholder variable
   DB_VAR7 : INT ;	//Temporary placeholder variable
   DB_VAR8 : INT ;	//Temporary placeholder variable
   DB_VAR9 : INT ;	//Temporary placeholder variable
   DB_VAR10 : INT ;	//Temporary placeholder variable
   DB_VAR11 : INT ;	//Temporary placeholder variable
   DB_VAR12 : INT ;	//Temporary placeholder variable
   DB_VAR13 : INT ;	//Temporary placeholder variable
   DB_VAR14 : INT ;	//Temporary placeholder variable
   DB_VAR15 : INT ;	//Temporary placeholder variable
   DB_VAR16 : INT ;	//Temporary placeholder variable
   DB_VAR17 : INT ;	//Temporary placeholder variable
   DB_VAR18 : INT ;	//Temporary placeholder variable
   DB_VAR19 : INT ;	//Temporary placeholder variable
   DB_VAR20 : INT ;	//Temporary placeholder variable
   DB_VAR21 : INT ;	//Temporary placeholder variable
   DB_VAR22 : INT ;	//Temporary placeholder variable
   DB_VAR23 : INT ;	//Temporary placeholder variable
   DB_VAR24 : INT ;	//Temporary placeholder variable
   DB_VAR25 : INT ;	//Temporary placeholder variable
   DB_VAR26 : INT ;	//Temporary placeholder variable
   DB_VAR27 : INT ;	//Temporary placeholder variable
   DB_VAR28 : INT ;	//Temporary placeholder variable
   DB_VAR29 : INT ;	//Temporary placeholder variable
   DB_VAR30 : INT ;	//Temporary placeholder variable
   DB_VAR31 : INT ;	//Temporary placeholder variable
   DB_VAR32 : INT ;	//Temporary placeholder variable
   DB_VAR33 : INT ;	//Temporary placeholder variable
   DB_VAR34 : INT ;	//Temporary placeholder variable
   DB_VAR35 : INT ;	//Temporary placeholder variable
   DB_VAR36 : INT ;	//Temporary placeholder variable
   DB_VAR37 : INT ;	//Temporary placeholder variable
   DB_VAR38 : INT ;	//Temporary placeholder variable
   DB_VAR39 : INT ;	//Temporary placeholder variable
   DB_VAR40 : INT ;	//Temporary placeholder variable
   DB_VAR41 : INT ;	//Temporary placeholder variable
   DB_VAR42 : INT ;	//Temporary placeholder variable
   DB_VAR43 : INT ;	//Temporary placeholder variable
   DB_VAR44 : INT ;	//Temporary placeholder variable
   DB_VAR45 : INT ;	//Temporary placeholder variable
   DB_VAR46 : INT ;	//Temporary placeholder variable
   DB_VAR47 : INT ;	//Temporary placeholder variable
   DB_VAR48 : INT ;	//Temporary placeholder variable
   DB_VAR49 : INT ;	//Temporary placeholder variable
   DB_VAR50 : INT ;	//Temporary placeholder variable
   DB_VAR51 : INT ;	//Temporary placeholder variable
   DB_VAR52 : INT ;	//Temporary placeholder variable
   DB_VAR53 : INT ;	//Temporary placeholder variable
   DB_VAR54 : INT ;	//Temporary placeholder variable
   DB_VAR55 : INT ;	//Temporary placeholder variable
   DB_VAR56 : INT ;	//Temporary placeholder variable
   DB_VAR57 : INT ;	//Temporary placeholder variable
   DB_VAR58 : INT ;	//Temporary placeholder variable
   DB_VAR59 : INT ;	//Temporary placeholder variable
   DB_VAR60 : INT ;	//Temporary placeholder variable
   DB_VAR61 : INT ;	//Temporary placeholder variable
   DB_VAR62 : INT ;	//Temporary placeholder variable
   DB_VAR63 : INT ;	//Temporary placeholder variable
   DB_VAR64 : INT ;	//Temporary placeholder variable
   DB_VAR65 : INT ;	//Temporary placeholder variable
   DB_VAR66 : INT ;	//Temporary placeholder variable
   DB_VAR67 : INT ;	//Temporary placeholder variable
   DB_VAR68 : INT ;	//Temporary placeholder variable
   DB_VAR69 : INT ;	//Temporary placeholder variable
   DB_VAR70 : INT ;	//Temporary placeholder variable
   DB_VAR71 : INT ;	//Temporary placeholder variable
   DB_VAR72 : INT ;	//Temporary placeholder variable
   DB_VAR73 : INT ;	//Temporary placeholder variable
   DB_VAR74 : INT ;	//Temporary placeholder variable
   DB_VAR75 : INT ;	//Temporary placeholder variable
   DB_VAR76 : INT ;	//Temporary placeholder variable
   DB_VAR77 : INT ;	//Temporary placeholder variable
   DB_VAR78 : INT ;	//Temporary placeholder variable
   DB_VAR79 : INT ;	//Temporary placeholder variable
   DB_VAR80 : INT ;	//Temporary placeholder variable
   DB_VAR81 : INT ;	//Temporary placeholder variable
   DB_VAR82 : INT ;	//Temporary placeholder variable
   DB_VAR83 : INT ;	//Temporary placeholder variable
   DB_VAR84 : INT ;	//Temporary placeholder variable
   DB_VAR85 : INT ;	//Temporary placeholder variable
   DB_VAR86 : INT ;	//Temporary placeholder variable
   DB_VAR87 : INT ;	//Temporary placeholder variable
   DB_VAR88 : INT ;	//Temporary placeholder variable
   DB_VAR89 : INT ;	//Temporary placeholder variable
   DB_VAR90 : INT ;	//Temporary placeholder variable
   DB_VAR91 : INT ;	//Temporary placeholder variable
   DB_VAR92 : INT ;	//Temporary placeholder variable
   DB_VAR93 : INT ;	//Temporary placeholder variable
   DB_VAR94 : INT ;	//Temporary placeholder variable
   DB_VAR95 : INT ;	//Temporary placeholder variable
   DB_VAR96 : INT ;	//Temporary placeholder variable
   DB_VAR97 : INT ;	//Temporary placeholder variable
   DB_VAR98 : INT ;	//Temporary placeholder variable
   DB_VAR99 : INT ;	//Temporary placeholder variable
   DB_VAR100 : INT ;	//Temporary placeholder variable
   DB_VAR101 : INT ;	//Temporary placeholder variable
   DB_VAR102 : INT ;	//Temporary placeholder variable
   DB_VAR103 : INT ;	//Temporary placeholder variable
   DB_VAR104 : INT ;	//Temporary placeholder variable
   DB_VAR105 : INT ;	//Temporary placeholder variable
   DB_VAR106 : INT ;	//Temporary placeholder variable
   DB_VAR107 : INT ;	//Temporary placeholder variable
   DB_VAR108 : INT ;	//Temporary placeholder variable
   DB_VAR109 : INT ;	//Temporary placeholder variable
   DB_VAR110 : INT ;	//Temporary placeholder variable
   DB_VAR111 : INT ;	//Temporary placeholder variable
   DB_VAR112 : INT ;	//Temporary placeholder variable
   DB_VAR113 : INT ;	//Temporary placeholder variable
   DB_VAR114 : INT ;	//Temporary placeholder variable
  END_STRUCT ;	
BEGIN
END_DATA_BLOCK

DATA_BLOCK "DB_HMI_Wozek"	// DB 128
AUTHOR : Kng
NAME : HMI_WOZ
VERSION : 0.1
  STRUCT
   HMI_IN : STRUCT 	//Zmienne wchodzace do HMI nie nadpisywane W HMI (100 bajtow) PLC-->HMI
    Komunikacja_Wozek_OK : BOOL ;	//### Komunikacja z wozkiem ok
    Wozek_W_Trybie_Auto : BOOL ;	//### Wozek znajduje sie w trybie auto
    Wozek_W_Trybie_Recznym : BOOL ;	//### Wozek znajduje sie w trybie recznym
    Wozek_Petla_0_OK : BOOL ;	//Petla bezpieczenstwa wozka ok
    Wozek_Petla_1_Ok : BOOL ;	//Petla bezpieczenstwa wozka ok
    Wozek_Zasprzeglony : BOOL ;	//### Wozek jest zasprzeglony z banda
    Wozek_Rozprzeglony : BOOL ;	//Wozek jest rozprzeglony z banda
    Wozek_Jest_W_Bledzie : BOOL ;	//### Wozek ma blad
    Pozycja_We_WY_KB1 : BOOL ;
    Pozycja_We_Wy_KB2 : BOOL ;
    Pozycja_We_Wy_Buffory : BOOL ;
    Pozycja_We_Wy_Gender : BOOL ;
    Rezerwa_191 : BOOL ;
    Rezerwa_1101 : BOOL ;
    Wozek_Banda_Lewo : BOOL ;
    Wozek_Banda_Prawo : BOOL ;
    Blokada_Intro_Aktywna : BOOL ;	//Blokada Intro aktywna
    Rezerwa_1141 : BOOL ;
    Rezerwa_1151 : BOOL ;
    Rezerwa_1161 : BOOL ;
    Rezerwa_112 : BOOL ;
    Rezerwa_113 : BOOL ;
    Rezerwa_114 : BOOL ;
    Rezerwa_115 : BOOL ;
    Wybrana_Strefa_1_Przod : BOOL ;	//Strefa 1 Skaner Przod (<--Shuttle) (dbx3.0)
    Wybrana_Strefa_2_Przod : BOOL ;	//Strefa 2 Skaner Przod (<--Shuttle)
    Wybrana_Strefa_3_Przod : BOOL ;	//Strefa 3 Skaner Przod (<--Shuttle)
    Wybrana_Strefa_4_Przod : BOOL ;	//Strefa 4 Skaner Przod (<--Shuttle)
    Wybrana_Strefa_1_Tyl : BOOL ;	//Strefa 1 Skaner Tyl(<--Shuttle)
    Wybrana_Strefa_2_Tyl : BOOL ;	//Strefa 2 Skaner Tyl (<--Shuttle)
    Wybrana_Strefa_3_Tyl : BOOL ;	//Strefa 3 Skaner Tyl (<--Shuttle)
    Wybrana_Strefa_4_Tyl : BOOL ;	//Strefa 4 Skaner Tyl (<--Shuttle)
    Pozycja_Aktualna : DINT ;	//###
    Rezerwa_222 : BOOL ;
    rezerwa_int : INT ;
    Nr_Bledu_Sew : INT ;	//Blad specyficzny sew do odczytania
    Prad_Aktualny : INT ;	//Prad aktualny SEW
    Predkosc_Aktualna_Wozek : INT ;	//Predkosc akutualna wozka
    Wartosc_Iteracji_Petli : INT ;
    Tablica_IN_INT : ARRAY  [1 .. 18 ] OF INT ;
    Tablica_IN_DWORD : ARRAY  [1 .. 9 ] OF DINT ;
    Aktualna_Data : DATE_AND_TIME ;
   END_STRUCT ;
   HMI_OUT : STRUCT 	//Zmienne wychodzace z HMI Nie nadpisywane w sterowniku (od 100 bajta ) HMI-->PLC
    rezerwaa : BOOL ;
    Przycisk_Wozek_Auto : BOOL ;	//Przycisk wozek auto (dbx100.1)
    Przycisk_Wozek_Reczny : BOOL ;	//Przycisk wozek reczny
    Przycisk_Wozek_Reset : BOOL ;	//Reset bledow wozek
    Przycisk_Wozek_Stop : BOOL ;	//Zatrzymanie zadania wozka
    Reset_Bledow : BOOL ;	//Reset bledow maszyny
    Reserwa_16 : BOOL ;
    Ladunek_Na_Intro : BOOL ;
    Reserwa122 : BOOL ;
    reserwa123 : BOOL ;
    Reserwa_110 : BOOL ;
    Reserwa_111 : BOOL ;
    Reserwa_112 : BOOL ;
    Reserwa_113 : BOOL ;
    reserwa : BOOL ;
    reserwa1 : BOOL ;
    Blokada_Pob_Intro : BOOL ;	//Zablokowaniec pobierania z intro
    Pozycja_Rezerwa : DINT ;
    Jedz_Na_Pozycje_KB1 : BOOL ;	//###
    Jedz_Na_Pozycje_KB2 : BOOL ;	//###
    Jedz_Na_Pozycje_Gender : BOOL ;	//###
    Jedz_Na_Pozycje_Odbior : BOOL ;	//###
    Jedz_Na_Pozycje_Pob_I1 : BOOL ;	//###
    Jedz_Na_Pozycje_Zadana : BOOL ;	//###
    Jedz_Na_Pozycje_Pob_I2 : BOOL ;
    Jedz_Na_Pozycje_Pob_I3 : BOOL ;
    r12 : BOOL ;
    r13 : BOOL ;
    r14 : BOOL ;
    r15 : BOOL ;
    r16 : BOOL ;
    r17 : BOOL ;
    r18 : BOOL ;
    r19 : BOOL ;
    Pozycja_5_Down : BOOL ;	//(dbx105.0)
    Pozycja_4_Up : BOOL ;
    Pozycja_4_Down : BOOL ;
    Pozycja_3_Up : BOOL ;
    Pozycja_3_Down : BOOL ;
    Pozycja_2_Up : BOOL ;
    Pozycja_2_Down : BOOL ;
    Pozycja_1_Up : BOOL ;
    r20 : BOOL ;
    Wartosc_Stosu_Elem_5 : INT ;
    Wartosc_Stosu_Elem_4 : INT ;
    Wartosc_Stosu_Elem_3 : INT ;
    Wartosc_Stosu_Elem_2 : INT ;
    Wartosc_Stosu_Elem_1 : INT ;
    Wartosc_Akutalnego_Kursu : INT ;
    r21 : BOOL ;
    r211 : BOOL ;
    r212 : BOOL ;
    r213 : BOOL ;
    r214 : BOOL ;
    r215 : BOOL ;
    r216 : BOOL ;
    r217 : BOOL ;
    r218 : BOOL ;
    r219 : BOOL ;
    r2110 : BOOL ;
    r2111 : BOOL ;
    r2112 : BOOL ;
    r2113 : BOOL ;
    r2114 : BOOL ;
    Reset_Para : BOOL ;
    PB_Default_Kier_KB1 : BOOL ;	//przycisk default kierunek rot-kb1
    PB_Move_Default_Kier_KB1 : BOOL ;	//Przycisk przesuwa wartosci z bloku 800 do 801
    PB_Write_Kier_KB1 : BOOL ;	//przycisk zapisania wartosc
    PB_Read_Kier_KB1 : BOOL ;	//przycisk odczytu wartosci
    PB_Move_Read_Kier_KB1 : BOOL ;	//przesuwa wartosc z db802 do db801
    PB_Save_Default_Kier_KB1 : BOOL ;	//zapisz do defaultowych
    Aktywny_Ekran_Kier_KB1 : BOOL ;
    res_kier_Kb11 : BOOL ;
    PB_Default_Kier_Rot : BOOL ;	//przycisk default kierunek
    PB_Move_Default_Kier_Rot : BOOL ;	//Przycisk przesuwa wartosci z bloku 800 do 801
    PB_Write_Kier_Rot : BOOL ;	//przycisk zapisania wartosc
    PB_Read_Kier_Rot : BOOL ;	//przycisk odczytu wartosci
    PB_Move_Read_Kier_Rot : BOOL ;	//przesuwa wartosc z db802 do db801
    PB_Save_Default_Kier_Rot : BOOL ;	//zapisuje do defaulta
    Aktywny_Ekran_Kier_Rot : BOOL ;
    res_kier_Kb13 : BOOL ;
    PB_Default_Para : BOOL ;	//przycisk default kierunek
    PB_Move_Default_Para : BOOL ;	//Przycisk przesuwa wartosci z bloku 800 do 801
    PB_Write_Para : BOOL ;	//przycisk zapisania wartosc
    PB_Read_Para : BOOL ;	//przycisk odczytu wartosci
    PB_Move_Read_Para : BOOL ;	//przesuwa wartosc z db802 do db801
    PB_Save_Default_Para : BOOL ;	//zapisuje parametry do defaultu
    Aktywny_Ekran_Kier_Para : BOOL ;
    res_kier_Kb15 : BOOL ;
    reserwa_int_1 : INT ;	//Wartosc iteracji wymienianych danych
    PB_Default_Odb : BOOL ;	//przycisk default kierunek
    PB_Move_Default_Odb : BOOL ;	//Przycisk przesuwa wartosci z bloku 800 do 801
    PB_Write_Odb : BOOL ;	//przycisk zapisania wartosc
    PB_Read_Odb : BOOL ;	//przycisk odczytu wartosci
    PB_Move_Read_Odb : BOOL ;	//przesuwa wartosc z db802 do db801
    PB_Save_Default_Odb : BOOL ;	//zapisuje parametry do defaultu
    Aktywny_Ekran_Odb : BOOL ;
    res_kier_Kb151 : BOOL ;
    Tablica_OUT_INT : ARRAY  [1 .. 12 ] OF INT ;
    Maska_Zadania : INT ;
    Tablica_OUT_DWORD : ARRAY  [1 .. 7 ] OF DWORD ;
    Reserwa_DWORD : DWORD ;
    Aktualna_Data : DATE_AND_TIME ;
   END_STRUCT ;
   HMI_IN_OUT : STRUCT 	//Zmienne nadpisywane w sterowniku i w HMI od 200 bajta
    Reserwa_in_out : BOOL ;
    rez_int : INT ;
    Pozycja_Zadana : DINT ;	//### Pozycja zadawana z HMI lub zadawana z PLC (dbd204)
    Wartosc_Buforu_Wozek : DINT ;
    Wartosc_Wozek_HMI : DINT ;	//Wartosc wozek dla HMI
    Wartosc_Wozek_HMI_HMI : DINT ;	//Wartosc wozek dla HMI
    Tablica_IN_OUT_INT : ARRAY  [1 .. 20 ] OF INT ;
    Tablica_IN_OUT_DWORD : ARRAY  [1 .. 8 ] OF DWORD ;
    Aktualna_Data : DATE_AND_TIME ;
   END_STRUCT ;
  END_STRUCT ;	
BEGIN
END_DATA_BLOCK

